fb_Product_Vacuum_Outlet_Isolation_Valve(Input1:= u01.product_vacuum_outlet_isolation_valve, Input2:= u.product_vacuum_outlet_isolation_valve, Output=> u01.XV_05);
u01.product_vacuum_outlet_isolation_valve_open_cmd_status				:= u01.XV_05;
u.product_vacuum_outlet_isolation_valve_clear							:= F_ValveClear(u.product_vacuum_outlet_isolation_valve, u01.product_vacuum_outlet_isolation_valve_open, u01.product_vacuum_outlet_isolation_valve_closed);

fb_Steam_Bypass_Valve(Input1:= u01.steam_bypass_valve, Input2:= u.steam_bypass_valve, Output=> u01.XV_08);
u01.steam_bypass_valve_open_cmd_status									:= u01.XV_08;
u.steam_bypass_valve_clear												:= F_ValveClear(u.steam_bypass_valve, u01.steam_bypass_valve_open, u01.steam_bypass_valve_closed);

fb_Condensate_Collection_Tank_Pump_Outlet_Valve(Input1:= u01.condensate_collection_tank_pump_outlet_valve, Input2:= u.condensate_collection_tank_pump_outlet_valve, Output=> );
u01.XV_09																:= u.condensate_collection_tank_pump_outlet_valve;
u01.condensate_collection_tank_pump_outlet_valve_open_cmd_status		:= u.condensate_collection_tank_pump_outlet_valve;
u.condensate_collection_tank_pump_outlet_valve_clear					:= F_ValveClear(u.condensate_collection_tank_pump_outlet_valve, u01.condensate_collection_tank_pump_outlet_valve_open, u01.condensate_collection_tank_pump_outlet_valve_closed);

fb_Product_Vacuum_Backfeed_Valve(Input1:= u01.product_vacuum_backfeed_valve, Input2:= u.product_vacuum_backfeed_valve);
fb_Product_Vacuum_Backfeed_Valve_Mode(Input1:= u01.product_vacuum_backfeed_valve_mode, Input2:= u.product_vacuum_backfeed_valve_mode);
fb_Product_Vacuum_Backfeed_Valve_PI(	Setpoint						:= u.product_vacuum_backfeed_valve_setpoint,
										Control							:= u01.product_vacuum_pres,
										Error							:= u01.product_vacuum_backfeed_valve_position_error,
										Reverse							:= FALSE,
										Kp								:= u01.product_vacuum_backfeed_valve_kp,           
										Ki								:= u01.product_vacuum_backfeed_valve_ki,           
										BaseAdjust						:= u01.product_vacuum_backfeed_valve_base_adjust,  
										LoopTime						:= u01.product_vacuum_backfeed_valve_loop_time,    
										IBand							:= u01.product_vacuum_backfeed_valve_iband,        
										Base							:= u01.product_vacuum_backfeed_valve_base,         
										Mode							:= u01.product_vacuum_backfeed_valve_mode,
										Input							:= u01.product_vacuum_backfeed_valve,
										Mode_Out						=> u01.product_vacuum_backfeed_valve_current_mode, 
										Output							=> u01.PCV_01);

u01.product_vacuum_backfeed_valve_position								:= INT_TO_REAL(u01.PCV_01_position) / _PERCENT_FACTOR; 
u.product_vacuum_backfeed_valve_open									:= u01.product_vacuum_backfeed_valve_position >= _VALVE_OPEN;
u01.product_vacuum_backfeed_valve_open									:= u.product_vacuum_backfeed_valve_open;
u.product_vacuum_backfeed_valve_closed									:= u01.product_vacuum_backfeed_valve_position < _VALVE_CLOSED;
u01.product_vacuum_backfeed_valve_closed								:= u.product_vacuum_backfeed_valve_closed;

fbSteamTotalizerEnable(Input1 := u01.steam_header_volume_total_enable, Input2 := u.steam_header_volume_total_enable );
//u01.steam_header_volume_total_enable 									:= u.steam_header_volume_total_enable;

fb_Product_Vacuum_Pump(					Enable							:= u01.product_vacuum_pump_vfd_enable,
										Pump_Reset						:= u01.product_vacuum_pump_reset,
										Purge_Time						:= u01.SP_product_vacuum_purge_time,
										Safety1							:= u01.P02_TSH_1,
										Safety2							:= u01.P02_TSH_2,
										Safety3							:= u01.P02_TSH_3,
										Error							=> u01.product_vacuum_pump_error,
										Purge_Solenoid_Valve			=> u01.P02_SVC_1,
										Seal_Purge_Valve				=> u01.P02_SVC_3);

sVacPumpError															:= CONCAT(gsProductVacuumPumpError, sVacuumPumpError[u01.product_vacuum_pump_error]);
bProductVacuumPumpError													:= P_Alarms.M_Check_Error(u01.product_vacuum_pump_error <> 0, bProductVacuumPumpError, _U01, sVacPumpError, gsProcessCannotRun);
						
fb_Product_Vacuum_Pump_Vfd_Input(Input1:= u01.product_vacuum_pump_vfd, Input2:= u.product_vacuum_pump_vfd);
rRpm																	:= u.product_vacuum_pump_vfd * _PUMP_RPM_FACTOR;
fb_Product_Vacuum_Pump_Vfd(				Enable_Vfd						:= fb_Product_Vacuum_Pump.Pump_On,
										Fault_Reset						:= u01.product_vacuum_pump_vfd_reset,
										Rpm								:= rRpm,
										Minimum_Speed					:= _PUMP_RPM_FACTOR * u01.SP_product_vacuum_idle_vfd_percent,
										Maximum_Speed					:= _PUMP_SPEED_MAX, 
										StatusWord						:= u01.product_vacuum_pump_vfd_status,
										ControlWord						=> u01.product_vacuum_pump_vfd_control, 
										TargetRpm						=> u01.product_vacuum_pump_vfd_target_vel, 
										Ready							=> u01.product_vacuum_pump_vfd_enabled,
										Error							=> u01.product_vacuum_pump_vfd_error);
u01.product_vacuum_pump_vfd_output  									:= WORD_TO_REAL(u01.product_vacuum_pump_vfd_velocity) / _PUMP_RPM_FACTOR ;                             
u.product_vacuum_pump_vfd_output										:= WORD_TO_REAL(u01.product_vacuum_pump_vfd_velocity);
IF u01.product_vacuum_pump_vfd_reset THEN
	u01.product_vacuum_pump_vfd_reset := FALSE;
END_IF

fb_Product_Vacuum_Pump_Radiator(Input1:= u01.radiator, Input2:= u.product_vacuum_pump_radiator);
u01.R_01																:= u.product_vacuum_pump_radiator;
u01.radiator_cmd_status													:= u.product_vacuum_pump_radiator;

// ignore if < 2 Amps
u01.l1_current_480														:= SEL(u01.IT_01 > _CURRENT_480_FACTOR * 2,0,F_IEConvert(u01.IT_01, _CURRENT_480_FACTOR));
u01.l2_current_480														:= SEL(u01.IT_02 > _CURRENT_480_FACTOR * 2,0,F_IEConvert(u01.IT_02, _CURRENT_480_FACTOR));
u01.l3_current_480														:= SEL(u01.IT_03 > _CURRENT_480_FACTOR * 2,0,F_IEConvert(u01.IT_03, _CURRENT_480_FACTOR));
u01.l1_voltage_480														:= F_IEConvert(u01.VT_01, _VOLTAGE_480_FACTOR);
u01.l2_voltage_480														:= F_IEConvert(u01.VT_02, _VOLTAGE_480_FACTOR);
u01.l3_voltage_480														:= F_IEConvert(u01.VT_03, _VOLTAGE_480_FACTOR);

// Ignore if < 1 Amp
u01.l1_current_208														:= SEL(u01.IT_04 > _CURRENT_208_FACTOR ,0,F_IEConvert(u01.IT_04, _CURRENT_208_FACTOR));
u01.l2_current_208														:= SEL(u01.IT_05 > _CURRENT_208_FACTOR ,0,F_IEConvert(u01.IT_05, _CURRENT_208_FACTOR));
u01.l3_current_208														:= SEL(u01.IT_06 > _CURRENT_208_FACTOR ,0,F_IEConvert(u01.IT_06, _CURRENT_208_FACTOR));
u01.l1_voltage_208														:= F_IEConvert(u01.VT_04, _VOLTAGE_208_FACTOR);
u01.l2_voltage_208														:= F_IEConvert(u01.VT_05, _VOLTAGE_208_FACTOR);
u01.l3_voltage_208														:= F_IEConvert(u01.VT_06, _VOLTAGE_208_FACTOR);

// Boiler - ignore noise if < 5A = 400 counts

u01.l1_current_boiler := SEL(u01.IT_boiler_01 > 400, 0, F_IEConvert(u01.IT_boiler_01, _CURRENT_BOILER_FACTOR));  // double coiled 
u01.l2_current_boiler := SEL(u01.IT_boiler_02 > 400, 0, F_IEConvert(u01.IT_boiler_02, _CURRENT_BOILER_FACTOR));  // double coiled 
u01.l3_current_boiler := SEL(u01.IT_boiler_03 > 400, 0, F_IEConvert(u01.IT_boiler_03, _CURRENT_BOILER_FACTOR));  // double coiled 

u01.boiler_ready														:= NOT u.boiler_outlet_pres_error AND u.boiler_outlet_pres > u01.SP_target_boiler_pressure AND u.boiler_package;
u.boiler_ready															:= u01.boiler_ready OR sita_bits[10].1;

tonBoilerCheck(IN:= u01.warmup_complete AND NOT u01.boiler_ready, PT:= _TIMEOUT_WARMUP_RESET);
IF tonBoilerCheck.Q THEN
	u01.warmup_complete													:= FALSE;
END_IF

// These Utility errors prevent any new automated cycles from running
u.utility_error															:= SEL(NOT u.boiler_ready, '', gsBoilerError);
u.utility_error															:= SEL(bDeadAirLinePresError, u.utility_error, gsDeadAirLinePresSensorError);		
u.utility_error															:= SEL(bPreCondenserLinePresError, u.utility_error, gsPreCondenserLinePresSensorError);
u.utility_error															:= SEL(bProductVacuumPresError, u.utility_error, gsProductVacuumPresSensorError);
u.utility_error															:= SEL(bProductVacuumPumpError, u.utility_error, gsProductVacuumPumpError);
u.utility_error															:= SEL(bProductOutletCo2Error, u.utility_error, gsProductOutletCo2SensorError);
u.utility_error															:= SEL(bProductOutletVolumetricFlowError, u.utility_error, gsProductOutletVolumetricFlowSensorError);
u.utility_error															:= SEL(bSteamHeaderFlowError, u.utility_error, gsSteamHeaderFlowSensorError);
u.utility_error															:= SEL(bBoilerOutletTempError, u.utility_error, gsBoilerOutletTempSensorError);
u.utility_error															:= SEL(bBoilerOutletPresError, u.utility_error, gsBoilerOutletPresSensorError);
u.utility_error															:= SEL(bProductCondensateDrumLevelError, u.utility_error, gsProductCondensateDrumLevelSensorError);
u.utility_error															:= SEL(bCondensateCollectionTankLevelError, u.utility_error, gsCondensateCollectionTankLevelSensorError);
u.utility_error															:= SEL(bWeatherTempUnsafe, u.utility_error, gsOutsideTempRangeError);
u.utility_error															:= SEL(bProductOutletPresError, u.utility_error, gsProductOutletPresSensorError);
u.utility_error															:= SEL(bProductOutletTempError, u.utility_error, gsProductOutletTempSensorError);
u.utility_error															:= SEL(bDeadAirLineCo2Error, u.utility_error, gsDeadAirLineCo2SensorError);
u.utility_error															:= SEL(bDeadAirFlowError, u.utility_error, gsDeadAirFlowSensorError);
u.utility_error															:= SEL(bProductOutletH2oError, u.utility_error, gsProductOutletH2oSensorError);
u.utility_error															:= SEL(bProductOutletO2Error, u.utility_error, gsProductOutletO2SensorError);
u.utility_error															:= SEL(bCondensateCollectionTankPhError, u.utility_error, gsCondensateCollectionTankPhSensorError);
u.utility_error															:= SEL(bCondensateCollectionTankO2Error, u.utility_error, gsCondensateCollectionTankO2SensorError);
u.utility_error															:= SEL(bCondensateCollectionTankTurbidityError, u.utility_error, gsCondensateCollectionTankTurbiditySensorError);
u.utility_error															:= SEL(bPurgeProductLinePresError, u.utility_error, gsPurgeProductLinePresSensorError);
u.utility_error															:= SEL(bPostCondenserLinePresError, u.utility_error, gsPostCondenserLinePresSensorError);
u.utility_error															:= SEL(bPurgeProductLineTempError, u.utility_error, gsPurgeProductLineTempSensorError);
u.utility_error															:= SEL(bPreCondenserLineTempError, u.utility_error, gsPreCondenserLineTempSensorError);
u.utility_error															:= SEL(bPostCondenserLineTempError, u.utility_error, gsPostCondenserLineTempSensorError);
u.utility_error															:= SEL(bProductCondenserPumpOutletTempError, u.utility_error, gsProductCondenserPumpOutletTempSensorError);
u.utility_error															:= SEL(bCondensateCollectionTankTempError, u.utility_error, gsCondensateCollectionTankTempSensorError);
u.utility_error															:= SEL(bCondensateCollectionTankOutletLineTempError, u.utility_error, gsCondensateCollectionTankOutletLineTempSensorError);
u.utility_error															:= SEL(bInstrumentAirCompPresError, u.utility_error, gsInstrumentAirCompPresSensorError);
u.utility_error															:= SEL(bInstrumentAirCompTempError, u.utility_error, gsInstrumentAirCompTempSensorError);
u.utility_error															:= SEL(bProductCondensateValveError, u.utility_error, gsProductCondensateDrainValveError);
sUtilityError															:= u.utility_error;

//P_Alarms.M_Add_Alarm('Utility', sUtilityError, 'Cycles_Stoppe');

// These errors initiate a Safe Shutdown if automated cycles are running 
IF m01.tb_Auto_Mode_On AND NOT bSafeShutdown THEN																			// Safe Shutdown 1
	u.safe_shutdown_error_1												:= SEL(bProductVacuumPumpError, '', gsProductVacuumPumpError);
	u.safe_shutdown_error_1												:= SEL(bPreCondenserLinePresError, u.safe_shutdown_error_1, gsPreCondenserLinePresSensorError);
	u.safe_shutdown_error_1												:= SEL(bProductVacuumPresError, u.safe_shutdown_error_1, gsProductVacuumPresSensorError);
	u.safe_shutdown_error_1												:= SEL(bProductOutletCo2Error, u.safe_shutdown_error_1, gsProductOutletCo2SensorError);
	u.safe_shutdown_error_1												:= SEL(bProductOutletVolumetricFlowError, u.safe_shutdown_error_1, gsProductOutletCo2SensorError);
	IF u.safe_shutdown_error_1 <> '' THEN
		bSafeShutdown													:= TRUE;
	ELSE																													// Safe Shutdown 2
		u.safe_shutdown_error_2											:= SEL(bSteamHeaderFlowError, '', gsSteamHeaderFlowSensorError);
		u.safe_shutdown_error_2											:= SEL(bBoilerOutletPresError, u.safe_shutdown_error_2, gsBoilerOutletPresSensorError);
		u.safe_shutdown_error_2											:= SEL(bBoilerOutletTempError, u.safe_shutdown_error_2, gsBoilerOutletTempSensorError);
		u.safe_shutdown_error_2											:= SEL(NOT u.boiler_ready, u.safe_shutdown_error_2, gsBoilerError);
		u.safe_shutdown_error_2											:= SEL(P_M01.bSteamManifoldLinePresError, u.safe_shutdown_error_2, gsSteamManifoldLinePresSensorError);
		u.safe_shutdown_error_2											:= SEL(P_M01.bSteamTempNearRS01Error, u.safe_shutdown_error_2, gsSteamTempNearRS01SensorError);
		u.safe_shutdown_error_2											:= SEL(P_M01.bSteamTempNearRS03Error, u.safe_shutdown_error_2, gsSteamTempNearRS03SensorError);
		u.safe_shutdown_error_2											:= SEL(bProductCondensateDrumLevelError, u.safe_shutdown_error_2, gsProductCondensateDrumLevelSensorError);
		u.safe_shutdown_error_2											:= SEL(bCondensateCollectionTankLevelError, u.safe_shutdown_error_2, gsCondensateCollectionTankLevelSensorError);
		IF u.safe_shutdown_error_2 <> '' THEN
			bSafeShutdown												:= TRUE;
		END_IF
	END_IF
ELSIF NOT m01.tb_Auto_Mode_On THEN
	bSafeShutdown														:= FALSE;
	u.safe_shutdown_error_1												:= '';
	u.safe_shutdown_error_2												:= '';
END_IF
END_ACTION

ACTION A_Totalizers:
tmrTotalizers(IN := NOT tmrTotalizers.Q,PT := T#1S);
// get steam density every 1 sec  
IF tmrTotalizers.Q THEN
	
 // Steam volume
	FOR idxSteamTable := 1 TO 30 DO 
		IF u01.boiler_outlet_pres >= STEAM_TABLE[idxSteamTable][0] THEN
			rSteamDensity := STEAM_TABLE[idxSteamTable][1];
		END_IF
	END_FOR
	
    u01.steam_header_volume := rSteamDensity * (u01.steam_header_flow*1000)/60 * 1.0;  // density kg/l  * flow m3/min ( m3 = 1000l)  * 1 sec 
	IF u01.steam_header_volume_total_enable THEN
		u01.steam_header_volume_total := u01.steam_header_volume_total + u01.steam_header_volume;
	ELSE
		u01.steam_header_volume_total := 0;
	END_IF
	
	// Product flows 
	IF u01.product_outlet_mass_flow_total_enable OR u01.product_outlet_volumetric_flow_total_enable THEN 
		u01.product_outlet_mass_flow_total := u01.product_outlet_mass_flow_total + u01.product_outlet_mass_flow/60 * 1.0;  //  kg/min to kg/sec * 1 sec
		u01.product_outlet_volumetric_flow_total := u01.product_outlet_volumetric_flow_total + u01.product_outlet_volumetric_flow/60 * 1.0 ;  // l/min to t/sec  * 1 sec
	ELSE
		u01.product_outlet_mass_flow_total := 0;
		u01.product_outlet_volumetric_flow_total := 0;
	END_IF
	
	// Bolier Water flow 
	
	IF u01.tap_water_to_boiler_flow_total_enable THEN 
		u01.tap_water_to_boiler_flow_total := u01.tap_water_to_boiler_flow_total +  u01.tap_water_to_boiler_flow/60 * 1.0; // //  kg/min to kg/sec * 1 sec
	ELSE
		u01.tap_water_to_boiler_flow_total := 0;
	END_IF
 
END_IF
END_ACTION

ACTION A_Weather_Station:
// Phase 0 - A_Weather_Station
// Rev 1.00 - February 5, 2024

IF iWSFunction = 0 THEN																		// Modbus is not busy
	WS_Master.UnitID 													:= 1;				// Weather Station Modbus address
	wWSAddress															:= 8193;
	wWSQuantity															:= 1;
	iWSFunction															:= eWSReadRegs;
	// Get weather values here
	//	ZXI_2002														:= wMBPReadData[0];
	//	ZYI_2002														:= wMBPReadData[1];
ELSIF tonWSReset.Q THEN
	iWSFunction															:= eWSIdle;
END_IF
tonWSReset(IN:= iWSFunction > 0, PT:= _TIMEOUT_MODBUS);

CASE iWSFunction OF
	
	eWSIdle:
		WS_Master.Execute 												:= FALSE;
		
	eWSReadRegs:
		WS_Master.ReadRegs(		Quantity								:= wWSQuantity, 
								MBAddr									:= wWSAddress, 
								cbLength								:= SIZEOF(wWSReadData), 
								pMemoryAddr								:= ADR(wWSReadData), 
								Execute									:= TRUE, 
								Timeout									:= _TIMEOUT_MODBUS, 
								BUSY									=> bWSBusy, 
								Error									=> bWSError, 
								ErrorId									=> WS_Errors, 
								cbRead									=> uiWSRead);
			
		WS_Master.ReadRegs(BUSY=> bWSBusy);
		IF NOT WS_Master.BUSY THEN
			WS_Master.Execute 											:= FALSE;
			WS_Master.ReadRegs(BUSY=> bWSBusy);
			IF WS_Master.Error THEN
				WS_Master.ReadRegs();
			ELSE
				iWSFunction 											:= 0;			
			END_IF
		END_IF
	
	ELSE
		iWSFunction 													:= 0;
	
END_CASE
END_ACTION

ACTION A2_WarmUp:
// Phase 0 - P_U01.A2_WarmUp
// Rev 1.0 - April 4, 2024

CASE i2Step OF

	0:	;
		
	1:	
		sError															:= '';
		bComplete														:= FALSE;
		bRunSteamBypass													:= FALSE;
		u01.steam_bypass_complete										:= FALSE;
		IF NOT u01.warmup_complete THEN
			gsCycleStage												:= 'warm_up.initialize';							// 3
			IF u01.boiler_outlet_pres_error THEN
				sError													:= F_Concat3(_U01, gsCycleStage, gsBoilerError);
				i2Step													:= 80;
			ELSE
				i2Step													:= i2Step + 1;
			END_IF
		ELSE
			bComplete													:= TRUE;
			i2Step														:= 90;
		END_IF
		
	2:	
		u01.boiler_package												:= TRUE;											// 4
		gsCycleStage													:= 'warm_up.boiler_heating';						// 5
		u01.drainage_on													:= TRUE;											// 6
		bAdsorptionActive												:= FALSE;											// 7
		bAdsorptionTimer												:= FALSE;
		i2Step															:= SEL(u01.SP_adsorb_during_warmup, 20, i2Step + 1);	// 8

	3:
		iAxStep															:= 1;												// 8.a
		i2Step															:= i2Step + 1;

	4:	
		Ax_Process_Pre_Check();																								// 8.a																			
		IF bPreCheckDone THEN
			IF sError = '' THEN																								// 8.a.i
				P_M01_RS01.open_repres_valves							:= P_M01.bRS01;										// 8.b
				P_M01_RS02.open_repres_valves							:= P_M01.bRS02;
				P_M01_RS03.open_repres_valves							:= P_M01.bRS03;
				rTime													:= _VALVE_TIME;
				i2Step													:= i2Step + 1;
			ELSE
				P_Alarms.M_Add_Alarm(CONCAT(_U01, gsCycleStage), sError, gsWarmupWillContinueWOAdsorption);					// 8.a.ii
				i2Step													:= 20;
			END_IF
		END_IF
		
	5:
		bTimer															:= TRUE;
		bPass1															:= (P_M01.bRS01 AND P_M01_RS01.repres_valves_clear) OR NOT P_M01.bRS01;
		bPass2															:= (P_M01.bRS02 AND P_M01_RS02.repres_valves_clear) OR NOT P_M01.bRS02;
		bPass3															:= (P_M01.bRS03 AND P_M01_RS03.repres_valves_clear) OR NOT P_M01.bRS03;
		IF bPass1 AND bPass2 AND bPass3 THEN
			bTimer														:= FALSE;
			i2Step														:= i2Step + 1;
		ELSIF tonTimer.Q THEN
			bTimer														:= FALSE;
			//P_M01_RS01.close_repres_valves								:= TRUE;
			//P_M01_RS02.close_repres_valves								:= TRUE;
			//P_M01_RS03.close_repres_valves								:= TRUE;
			//P_Alarms.M_Add_Alarm(CONCAT(_U01, gsCycleStage), M_Repres_Valve_Error(), gsWarmupWillContinueWOAdsorption);	// Per Alex W.
			//i2Step														:= 20;
			i2Step														:= i2Step + 1; 
		END_IF
		
	6:
		P_M01_RS01.open_all_doors										:= P_M01.bRS01;										// 8.c
		P_M01_RS02.open_all_doors										:= P_M01.bRS02;
		P_M01_RS03.open_all_doors										:= P_M01.bRS03;
		rTime															:= m01.SP_doorsopenclose_timedelay * _MINUTES;										// 8.c.i
		gsCycleStage													:= 'warm_up.boiler_heating_open_doors';				// 8.c.ii
		i2Step															:= i2Step + 1;

	7:
		bTimer															:= TRUE; 
		bPass1															:= (P_M01.bRS01 AND P_M01_RS01.R_S.all_doors_open) OR NOT P_M01.bRS01;
		bPass2															:= (P_M01.bRS02 AND P_M01_RS02.R_S.all_doors_open) OR NOT P_M01.bRS02;
		bPass3															:= (P_M01.bRS03 AND P_M01_RS03.R_S.all_doors_open) OR NOT P_M01.bRS03;
		IF bPass1 AND bPass2 AND bPass3 THEN
			bTimer														:= FALSE;
			i2Step														:= i2Step + 1;
		ELSIF tonTimer.Q THEN
			bTimer														:= FALSE;
			sRS															:= SEL(NOT bPass1, SEL(NOT bPass2, _RS03, _RS02), _RS01);
			P_Alarms.M_Add_Alarm(F_Concat3(_U01, sRS, gsCycleStage), gsReactorDoorOpeningError, gsWarmupWillContinueWOAdsorption);
			i2Step														:= 20;
		END_IF

	8:
		P_M01_RS01.fan_vfd_percent										:= SEL(P_M01.bRS01, 0, m01.SP_reactor_set_1_vfd_percent);	// 8.d
		P_M01_RS02.fan_vfd_percent										:= SEL(P_M01.bRS02, 0, m01.SP_reactor_set_2_vfd_percent);
		P_M01_RS03.fan_vfd_percent										:= SEL(P_M01.bRS03, 0, m01.SP_reactor_set_3_vfd_percent);
		gsCycleStage													:= 'warm_up.boiler_heating_turn_on_fans';			// 8.d.i
		rTime															:= _FAN_RS_DELAY_TIME;
		i2Step															:= i2Step + 1;

	9:
		bTimer															:= TRUE;
		IF tonTimer.Q THEN
			bTimer														:= FALSE;
			i2Step														:= i2Step + 1;
		END_IF

	10:
		P_M01_RS01.co2_inside_sensors_on								:= P_M01.bRS01;										// 8.e
		P_M01_RS02.co2_inside_sensors_on								:= P_M01.bRS02;
		P_M01_RS03.co2_inside_sensors_on								:= P_M01.bRS03;
		gsCycleStage													:= 'warm_up.boiler_heating_adsorption';				// 8.e.i
		bAdsorptionTimer												:= TRUE;											// 8.f
		bAdsorptionActive												:= TRUE;											// 8.g
		i2Step															:= 20;


//**** Complete Warmup		
	20:
		u01.product_vacuum_backfeed_valve								:= _OPEN;											// 9
		rTime															:= _VALVE_TIME;
		i2Step															:= i2Step + 1;
		
	21:	
		bTimer															:= TRUE;
		IF u01.product_vacuum_backfeed_valve_open THEN																		// 9
			bTimer														:= FALSE;
			u01.product_vacuum_pump_vfd									:= u01.SP_product_vacuum_idle_vfd_percent;			// 10
			rTime														:= u01.SP_boiler_warmup_duration * _MINUTES;		// 11
			i2Step														:= i2Step + 1;
		ELSIF tonTimer.Q THEN
			bTimer														:= FALSE;
			sError														:= gsProductVacuumBackfeedValveError;				// 9
			IF bAdsorptionActive THEN
				P_Alarms.M_Add_Alarm(CONCAT(_U01, gsCycleStage), sError, gsProcessCannotRunAdsorptionWillContinue);
				u01.boiler_package										:= FALSE;
				i2Step													:= 30;
			ELSE
				i2Step													:= 80;
			END_IF
		END_IF
		
	22:
		bTimer															:= TRUE;
		IF u01.boiler_ready THEN																							// 12 (Handled in P_U01.A_Points)
			bTimer														:= FALSE;
			bComplete													:= TRUE;
			u01.warmup_complete											:= TRUE;
			i2Step														:= i2Step + 1;
		ELSIF tonTimer.Q THEN																								// 12.a
			bTimer														:= FALSE;
			sError														:= gsBoilerError;
			i2Step														:= 80;
		END_IF

	23:
		bRunSteamBypass													:= u01.SP_steam_bypass_immediately_after_warm_up;
		IF bAdsorptionActive AND NOT bRunSteamBypass THEN 																	// 14
			i2Step														:= 30;
		ELSIF bAdsorptionActive AND bRunSteamBypass AND NOT u01.SP_adsorb_during_steam_bypass THEN
			i2Step														:= 40;												// 15
		ELSE
			i2Step														:= 90;												// 13 & 16
		END_IF
	
		
//**** Adsorption 1		
	30:
		IF tonAdsorptionTimer.Q THEN																						// 14.a
			bAdsorptionTimer											:= FALSE;
			gsCycleStage												:= 'warm_up.boiler_heating.turn_off_fans';			// 14.b
			P_M01_RS01.fan_vfd_percent									:= 0;												// 14.c
			P_M01_RS02.fan_vfd_percent									:= 0;
			P_M01_RS03.fan_vfd_percent									:= 0;
			rTime														:= _FAN_RS_DELAY_TIME;
			i2Step														:= i2Step + 1;
		END_IF

	31:
		bTimer															:= TRUE;
		IF tonTimer.Q THEN
			bTimer														:= FALSE;
			gsCycleStage												:= 'warm_up.boiler_heating.closing_doors';			// 14.d
			P_M01_RS01.close_all_doors									:= TRUE;											// 14.e
			P_M01_RS02.close_all_doors									:= TRUE;
			P_M01_RS03.close_all_doors									:= TRUE;
			rTime														:= m01.SP_doorsopenclose_timedelay * _MINUTES;										// 14.e.i
			i2Step														:= i2Step + 1;
		END_IF		

	32:
		bTimer															:= TRUE;
		bPass1															:= (P_M01.bRS01 AND P_M01_RS01.R_S.all_doors_closed) OR NOT P_M01.bRS01;	// 14.e.ii
		bPass2															:= (P_M01.bRS02 AND P_M01_RS02.R_S.all_doors_closed) OR NOT P_M01.bRS02;
		bPass3															:= (P_M01.bRS03 AND P_M01_RS03.R_S.all_doors_closed) OR NOT P_M01.bRS03;
		IF bPass1 AND bPass2 AND bPass3 THEN
			bTimer														:= FALSE;
			i2Step														:= i2Step + 1;
		ELSIF tonTimer.Q THEN																								// 14.e.i
			bTimer														:= FALSE;
			bRunSteamBypass												:= FALSE;
			sRS															:= SEL(NOT bPass1, SEL(NOT bPass2, _RS03, _RS02), _RS01);
			P_Alarms.M_Add_Alarm(F_Concat3(_U01, sRS, gsCycleStage), gsReactorDoorClosingError, gsSystemCannotRun);
			i2Step														:= i2Step + 1;
		END_IF
		
	33:
		P_M01_RS01.co2_sensors_off										:= TRUE;											// 14.f
		P_M01_RS02.co2_sensors_off										:= TRUE;
		P_M01_RS03.co2_sensors_off										:= TRUE;
		bAdsorptionActive												:= FALSE;											// 14.g
		i2Step															:= 90;

	
//**** Adsorption 2	
	40:
		IF tonAdsorptionTimer.Q THEN																						// 15.a
			bAdsorptionTimer											:= FALSE;
			P_M01_RS01.fan_vfd_percent									:= 0;												// 15.b
			P_M01_RS02.fan_vfd_percent									:= 0;
			P_M01_RS03.fan_vfd_percent									:= 0;
			rTime														:= _FAN_RS_DELAY_TIME;
			i2Step														:= i2Step + 1;
		END_IF

	41:
		bTimer															:= TRUE;
		IF tonTimer.Q THEN
			bTimer														:= FALSE;											// 15.c
			P_M01_RS01.co2_sensors_off									:= TRUE;
			P_M01_RS02.co2_sensors_off									:= TRUE;
			P_M01_RS03.co2_sensors_off									:= TRUE;
			bAdsorptionActive											:= FALSE;											// 15.d
			i2Step														:= i2Step + 1;
		END_IF
		
	42:
		P_M01_RS01.close_all_doors										:= TRUE;											// 15.g
		P_M01_RS02.close_all_doors										:= TRUE;
		P_M01_RS03.close_all_doors										:= TRUE;
		rTime															:= m01.SP_doorsopenclose_timedelay * _MINUTES;										// 15.g.i
		i2Step															:= i2Step + 1;

	43:
		bTimer															:= TRUE;
		bPass1															:= (P_M01.bRS01 AND P_M01_RS01.R_S.all_doors_closed) OR NOT P_M01.bRS01;		// 15.g.ii
		bPass2															:= (P_M01.bRS02 AND P_M01_RS02.R_S.all_doors_closed) OR NOT P_M01.bRS02;
		bPass3															:= (P_M01.bRS03 AND P_M01_RS03.R_S.all_doors_closed) OR NOT P_M01.bRS03;
		IF bPass1 AND bPass2 AND bPass3 THEN
			bTimer														:= FALSE;
			i2Step														:= 90;
		ELSIF tonTimer.Q THEN
			bTimer														:= FALSE;
			bRunSteamBypass												:= FALSE;
			sRS															:= SEL(NOT bPass1, SEL(NOT bPass2, _RS03, _RS02), _RS01);
			P_Alarms.M_Add_Alarm(F_Concat3(_U01, sRS, gsCycleStage), gsReactorDoorOpeningError, gsSystemCannotRun);
			i2Step														:= 90;
		END_IF


//**** Process error		
	80:
		P_Alarms.M_Add_Alarm(CONCAT(_U01, gsCycleStage), sError, gsProcessCannotRun);
		gsCycleStage													:= 'warm_up.error';
		i2Step															:= i2Step + 1;

//**** Stop process		
	81:
		u01.product_vacuum_pump_vfd										:= 0;
		u01.product_vacuum_backfeed_valve								:= _CLOSED;
		P_M01_RS01.co2_sensors_off										:= TRUE;
		P_M01_RS02.co2_sensors_off										:= TRUE;
		P_M01_RS03.co2_sensors_off										:= TRUE;
		P_M01_RS01.fan_vfd_percent										:= 0;
		P_M01_RS02.fan_vfd_percent										:= 0;
		P_M01_RS03.fan_vfd_percent										:= 0;
		rTime															:= _FAN_RS_DELAY_TIME;
		i2Step															:= i2Step + 1;

	82:
		bTimer															:= TRUE;
		IF tonTimer.Q THEN
			bTimer														:= FALSE;
			u01.boiler_package											:= FALSE;
			P_M01_RS01.close_all_doors									:= P_M01.bRS01;
			P_M01_RS02.close_all_doors									:= P_M01.bRS02;
			P_M01_RS03.close_all_doors									:= P_M01.bRS03;
			rTime														:= m01.SP_doorsopenclose_timedelay * _MINUTES;
			i2Step														:= 90;
		END_IF
		
//**** Close process
	90:
		gsCycleStage													:= SEL(bComplete, 'warm_up.failed', 'warm_up.complete');
		bAdsorptionTimer												:= FALSE;
		u01.drainage_on													:= FALSE;
		rTime															:= _PROCESS_COMPLETE_TIME;
		i2Step															:= i2Step + 1;
		
	91:
		bTimer															:= TRUE;
		IF tonTimer.Q THEN
			bTimer														:= FALSE;
			gsCycleStage												:= '';
			i2Step														:= 0;
		END_IF
				

END_CASE

IF i2Step > 0 AND i2Step < 80 AND u01.shutdown_process THEN
	gsCycleStage														:= 'warm_up.stopping';
	i2Step																:= 81;
END_IF
END_ACTION

ACTION A3_Steam_Bypass:
// Phase 0 - P_U01.A3_Steam_Bypass
// Rev 1.0 - April 4, 2024

CASE i3Step OF

	0:	;

	1:	
		bComplete														:= FALSE;
		IF u01.warmup_complete THEN
			IF NOT u01.steam_bypass_complete THEN
				gsCycleStage											:= 'steam_bypass.initialize';						// 4
				sError													:= '';
				IF u01.post_condenser_line_pres_error THEN
					sError												:= gsPostCondenserLinePresSensorError;
				ELSIF u01.pre_condenser_line_pres_error THEN
					sError												:= gsPreCondenserLinePresSensorError;
				ELSIF u01.purge_product_line_pres_error THEN
					sError												:= gsPurgeProductLinePresSensorError;
				ELSIF u01.product_vacuum_pres_error THEN
					sError												:= gsProductVacuumPresSensorError;
				ELSIF u01.steam_header_flow_error THEN
					sError												:= gsSteamHeaderFlowSensorError;
				ELSIF u01.purge_product_line_temp_error THEN
					sError												:= gsPurgeProductLineTempSensorError;
				END_IF
				i3Step													:= SEL(sError = '', 80, i3Step + 1);
			ELSE
				bComplete												:= TRUE;
				i3Step													:= 90;
			END_IF
		ELSE
			u01.boiler_package											:= FALSE;
			P_Alarms.M_Add_Alarm(CONCAT(_U01, gsCycleStage), gsWarmupNotRunError, gsProcessCannotRun);
			i3Step														:= 90;
		END_IF
		
	2:	
		IF u01.boiler_ready THEN																							// 5.a (Handled in P_U01.A_Points)
			P_U01.bCloseXVValves										:= TRUE;											// 5.b
			rTime														:= _VALVE_TIME;
			i3Step														:= i3Step + 1;
		ELSE
			sError														:= gsBoilerError;
			sMessage													:= gsRunWarmup;
			i3Step														:= 80;
		END_IF

	3:	bTimer															:= TRUE;
		bPass1															:= u01.product_vacuum_pump_isolation_valve_closed;
		bPass2															:= u01.product_vacuum_outlet_isolation_valve_closed;
		IF bPass1 AND bPass2 THEN
			bTimer														:= FALSE;
			u01.product_vacuum_backfeed_valve							:= _OPEN;											// 5.b.iii
			rTime														:= _VALVE_TIME;
			i3Step														:= i3Step + 1;
		ELSIF tonTimer.Q THEN
			bTimer														:= FALSE;
			sError														:= SEL(bPass1, '', gsProductVacuumPumpIsoValveError);
			sError														:= SEL(bPass2, sError, gsProductVacuumOutletIsoValveError);
			i3Step														:= 80;
		END_IF
		
	4:
		bTimer															:= TRUE;
		IF u01.product_vacuum_backfeed_valve > _VALVE_OPEN THEN
			bTimer														:= FALSE;
			u01.drainage_on												:= TRUE;											// 5.c
			u01.product_vacuum_pump_vfd									:= u01.SP_product_vacuum_idle_vfd_percent;			// 5.d.ii
			IF bAdsorptionActive AND u01.SP_adsorb_during_steam_bypass THEN													// 5.b.iv
				P_M01_RS01.open_all_doors								:= P_M01.bRS01;
				P_M01_RS02.open_all_doors								:= P_M01.bRS02;
				P_M01_RS03.open_all_doors								:= P_M01.bRS03;
				rTime													:= m01.SP_doorsopenclose_timedelay * _MINUTES;
				i3Step													:= i3Step + 1;
			ELSE
				i3Step													:= i3Step + 2;
			END_IF
		ELSIF tonTimer.Q THEN
			bTimer														:= FALSE;
			sError														:= gsProductVacuumBackfeedValveError;
			i3Step														:= 80;
		END_IF

	5:
		bTimer															:= TRUE;
		bPass1															:= (P_M01.bRS01 AND P_M01_RS01.R_S.all_doors_open) OR NOT P_M01.bRS01;	// 5.b.iv
		bPass2															:= (P_M01.bRS02 AND P_M01_RS02.R_S.all_doors_open) OR NOT P_M01.bRS02;
		bPass3															:= (P_M01.bRS03 AND P_M01_RS03.R_S.all_doors_open) OR NOT P_M01.bRS03;
		IF bPass1 AND bPass2 AND bPass3 THEN
			bTimer														:= FALSE;
			IF NOT bAdsorptionActive AND u01.SP_adsorb_during_steam_bypass THEN												// 6
				iAxStep													:= 1;												// 6.b
				i3Step													:= i3Step + 1;
			ELSE
				i3Step													:= 20;
			END_IF
		ELSIF tonTimer.Q THEN
			bTimer														:= FALSE;
			bAdsorptionActive											:= FALSE;
			sRS															:= SEL(NOT bPass1, SEL(NOT bPass2, _RS03, _RS02), _RS01);
			P_Alarms.M_Add_Alarm(F_Concat3(_U01, sRS, gsCycleStage), gsReactorDoorOpeningError, gsSteamBypassWillContinueWOAdsorption);
			i3Step														:= 20;
		END_IF

	6:
		Ax_Process_Pre_Check();																								// 6.b																			
		IF bPreCheckDone THEN
			IF sError = '' THEN																								// 6.b.i
				P_M01_RS01.open_repres_valves							:= P_M01.bRS01;										// 6.c
				P_M01_RS02.open_repres_valves							:= P_M01.bRS02;
				P_M01_RS03.open_repres_valves							:= P_M01.bRS03;
				rTime													:= _VALVE_TIME;
				i3Step													:= i3Step + 1;
			ELSE
				P_Alarms.M_Add_Alarm(CONCAT(_U01, gsCycleStage), sError, gsSteamBypassWillContinueWOAdsorption);			// 6.b.ii
				bAdsorptionActive										:= FALSE;
				i3Step													:= 20;
			END_IF
		END_IF

	7:
		bTimer															:= TRUE;
		bPass1															:= (P_M01.bRS01 AND P_M01_RS01.repres_valves_clear) OR NOT P_M01.bRS01;
		bPass2															:= (P_M01.bRS02 AND P_M01_RS02.repres_valves_clear) OR NOT P_M01.bRS02;
		bPass3															:= (P_M01.bRS03 AND P_M01_RS03.repres_valves_clear) OR NOT P_M01.bRS03;
		IF bPass1 AND bPass2 AND bPass3 THEN
			bTimer														:= FALSE;
			i3Step														:= i3Step + 1;
		ELSIF tonTimer.Q THEN
			bTimer														:= FALSE;
			i3Step														:= i3Step + 1;
			//P_Alarms.M_Add_Alarm(CONCAT(_U01, gsCycleStage), M_Repres_Valve_Error(), gsSteamBypassWillContinueWOAdsorption);
			//bAdsorptionActive											:= FALSE;
			//P_M01_RS01.close_repres_valves								:= P_M01.bRS01;
			//P_M01_RS02.close_repres_valves								:= P_M01.bRS02;
			//P_M01_RS03.close_repres_valves								:= P_M01.bRS03;
			//i3Step													:= 20; 
		END_IF
		
	8:
		P_M01_RS01.open_all_doors										:= P_M01.bRS01;
		P_M01_RS02.open_all_doors										:= P_M01.bRS02;
		P_M01_RS03.open_all_doors										:= P_M01.bRS03;
		gsCycleStage													:= 'steam_bypass.initialize.open_doors';			// 6.d.ii
		rTime															:= m01.SP_doorsopenclose_timedelay * _MINUTES;										// 6.d.i
		i3Step															:= i3Step + 1;

	9:
		bTimer															:= TRUE; 
		bPass1															:= (P_M01.bRS01 AND P_M01_RS01.R_S.all_doors_open) OR NOT P_M01.bRS01;	// 6.d.ii
		bPass2															:= (P_M01.bRS02 AND P_M01_RS02.R_S.all_doors_open) OR NOT P_M01.bRS02;
		bPass3															:= (P_M01.bRS03 AND P_M01_RS03.R_S.all_doors_open) OR NOT P_M01.bRS03;
		IF bPass1 AND bPass2 AND bPass3 THEN
			bTimer														:= FALSE;
			i3Step														:= i3Step + 1;
		ELSIF tonTimer.Q THEN
			bTimer														:= FALSE;
			sRS															:= SEL(NOT bPass1, SEL(NOT bPass2, _RS03, _RS02), _RS01);
			P_Alarms.M_Add_Alarm(F_Concat3(_U01, sRS, gsCycleStage), gsReactorDoorOpeningError, gsSteamBypassWillContinueWOAdsorption);
			bAdsorptionActive											:= FALSE;
			i3Step														:= 20;
		END_IF

	10:
		P_M01_RS01.fan_vfd_percent										:= SEL(P_M01.bRS01, 0, m01.SP_reactor_set_1_vfd_percent);	// 6.e
		P_M01_RS02.fan_vfd_percent										:= SEL(P_M01.bRS02, 0, m01.SP_reactor_set_2_vfd_percent);
		P_M01_RS03.fan_vfd_percent										:= SEL(P_M01.bRS03, 0, m01.SP_reactor_set_3_vfd_percent);
		gsCycleStage													:= 'steam_bypass.initialize.turn_on_fans';			// 6.e.i
		rTime															:= _FAN_RS_DELAY_TIME;
		i3Step															:= i3Step + 1;

	11:
		bTimer															:= TRUE;
		IF tonTimer.Q THEN
			bTimer														:= FALSE;
			i3Step														:= i3Step + 1;
		END_IF

	12:
		P_M01_RS01.co2_inside_sensors_on								:= P_M01.bRS01;										// 6.f
		P_M01_RS02.co2_inside_sensors_on								:= P_M01.bRS02;
		P_M01_RS03.co2_inside_sensors_on								:= P_M01.bRS03;
		gsCycleStage													:= 'steam_bypass.initialize.adsorption';			// 6.f.i
		bAdsorptionTimer												:= TRUE;											// 6.a
		bAdsorptionActive												:= TRUE;											// 6.g
		i3Step															:= 20;


//**** Complete Steam Bypass		
	20:
		u01.product_condenser											:= TRUE;											// 7
		rSP																:= u01.SP_steam_bypass_vacuum_pressure;				// 8
		bPass1															:= u01.product_vacuum_pres < rSP;
		bPass2															:= u01.post_condenser_line_pres < rSP;
		bPass3															:= u01.pre_condenser_line_pres < rSP;
		bPass4															:= u01.purge_product_line_pres < rSP;
		i3Step															:= SEL(bPass1 AND bPass2 AND bPass3 AND bPass4, i3Step + 1, 30);
	
	21:
		u01.product_vacuum_pump_isolation_valve							:= TRUE;											// 9.a
		u01.product_vacuum_outlet_isolation_valve						:= TRUE;
		rTime															:= _VALVE_TIME;
		i3Step															:= i3Step + 1;
		
	22:
		bTimer															:= TRUE;
		bPass1															:= u01.product_vacuum_pump_isolation_valve_open;
		bPass2															:= u01.product_vacuum_outlet_isolation_valve_open;
		IF bPass1 AND bPass2 THEN
			bTimer														:= FALSE;
			//u01.product_blower											:= TRUE;											// 9.a
			u.product_blower_vfd										:= 0;  //
			u01.product_vacuum_backfeed_valve							:= _CLOSED;
			i3Step														:= i3Step + 1;
		ELSIF tonTimer.Q THEN
			bTimer														:= FALSE;
			sError														:= SEL(bPass1, '', gsProductVacuumPumpIsoValveError);
			sError														:= SEL(bPass2, sError, gsProductVacuumOutletIsoValveError);
			i3Step														:= 80;
		END_IF
		
	23:	
		u01.product_vacuum_pump_vfd										:= u01.SP_product_vacuum_running_vfd_percent;			// 9.b
		gsCycleStage													:= SEL(bAdsorptionActive, 'steam_bypass.evacuate_lines', 'steam_bypass.evacuate_lines.adsorption');		// 9.b.i
		u01.purge_product_pre_condenser_valve							:= TRUE;											// 9.c
		u01.cooling_line_pre_condenser_valve							:= TRUE;
		rTime															:= m01.SP_evacuation_duration * _MINUTES;
		i3Step															:= i3Step + 1;
		
	24:
		bTimer															:= TRUE;											// 9.d
		rSP																:= u01.SP_steam_bypass_vacuum_pressure;
		bPass1															:= u01.product_vacuum_pres < rSP;
		bPass2															:= u01.post_condenser_line_pres < rSP;
		bPass3															:= u01.pre_condenser_line_pres < rSP;
		bPass4															:= u01.purge_product_line_pres < rSP;
		IF bPass1 AND bPass2 AND bPass3 AND bPass4 THEN
			bTimer														:= FALSE;
			i3Step														:= i3Step + 1;
		ELSIF tonTimer.Q THEN
			bTimer														:= FALSE;
			sError														:= gsUnableToEvacuateLinesError;
			i3Step														:= 80;
		END_IF
	
	25:	
		u01.product_vacuum_pump_isolation_valve							:= FALSE;											// 9.e
		u01.product_vacuum_outlet_isolation_valve						:= FALSE;
		u01.product_vacuum_backfeed_valve								:= _OPEN;
		//u01.product_blower											:= FALSE;
		u.product_blower_vfd											:= 0;
		u01.cooling_line_pre_condenser_valve							:= FALSE;
		u01.purge_product_pre_condenser_valve							:= FALSE;
		u01.product_vacuum_pump_vfd										:= u01.SP_product_vacuum_idle_vfd_percent;			// 9.f
		i3Step															:= 30;

		
//**** Steam Bypass		
	30:
		u01.steam_bypass_valve											:= TRUE;											// 10
		gsCycleStage													:= SEL(bAdsorptionActive, 'steam_bypass.steam_bypass.adsorption', 'steam_bypass.steam_bypass');		// 10.a
		rSP																:= u01.SP_steam_bypass_duration * _MINUTES;				
		rTime															:= rSP;
		i3Step															:= i3Step + 1;				

	31:
		bTimer															:= TRUE;											// 10.b
		IF u01.purge_product_line_pres > m01.SP_steam_purge_pressure THEN													// 11
			i3Step														:= i3Step + 1;
		ELSIF tonTimer.Q THEN
			bTimer														:= FALSE;
			sError														:= gsPurgeProductLinePresLowError;
			i3Step														:= 80;
		END_IF
		
	32:
		u01.product_vacuum_bypass_valve									:= TRUE;											// 12
		u01.purge_product_pre_condenser_valve							:= TRUE;
		//u01.product_blower												:= TRUE;
		u.product_blower_vfd											:= _BLOWER_RPM_FACTOR * 100; // % TBD 
		i3Step															:= i3Step + 1;
		
	33:
		IF TIME_TO_REAL(tonTimer.ET) >= (rSP * 0.3) THEN																	// 13
			i3Step														:= i3Step + 1;
		END_IF 
	
	34:
		IF u01.steam_header_flow > u01.SP_minimum_steam_bypass_flow_rate THEN
			i3Step														:= i3Step + 1;										// 13.a
		ELSE
			sError														:= gsSteamBypassMinFlowRateError;					// 13.b
			i3Step														:= 80;
		END_IF
	
	35:
		IF tonTimer.Q OR u01.purge_product_line_temp > u01.SP_steam_bypass_temperature THEN									// 14
			bTimer														:= FALSE;
			u01.steam_bypass_valve										:= FALSE;											// 15
			gsCycleStage												:= SEL(bAdsorptionActive, 'steam_bypass.wrap_up', 'steam_bypass.wrap_up.adsorption');	// 15.a
			u01.purge_product_pre_condenser_valve						:= FALSE;											// 16
			u01.product_vacuum_bypass_valve								:= FALSE;
			u01.product_condenser										:= FALSE;
			//u01.product_blower											:= FALSE;
			u.product_blower_vfd										:= 0;
			IF bAdsorptionActive THEN
				i3Step													:= 40;
			ELSE
				u01.steam_bypass_complete								:= TRUE;
				i3Step													:= 90;
			END_IF
		END_IF
		
		
//**** Complete Adsorption		
	40:
		IF tonAdsorptionTimer.Q THEN																						// 17.a.i
			bAdsorptionTimer											:= FALSE;
			P_M01_RS01.fan_vfd_percent									:= 0;												// 17.a.ii
			P_M01_RS02.fan_vfd_percent									:= 0;
			P_M01_RS03.fan_vfd_percent									:= 0;
			gsCycleStage												:= 'steam_bypass.wrap_up.turn_off_fans';			// 17.a.ii.1
			rTime														:= _FAN_RS_DELAY_TIME;
			i3Step														:= i3Step + 1;
		END_IF

	41:
		bTimer															:= TRUE;
		IF tonTimer.Q THEN
			bTimer														:= FALSE;
			P_M01_RS01.close_all_doors									:= TRUE;											// 17.a.iii
			P_M01_RS02.close_all_doors									:= TRUE;
			P_M01_RS03.close_all_doors									:= TRUE;
			gsCycleStage												:= 'steam_bypass.wrap_up.close_doors';				// 17.a.iii.1
			rTime														:= m01.SP_doorsopenclose_timedelay * _MINUTES;										// 17.a.iii.2
			i3Step														:= i3Step + 1;
		END_IF		

	42:
		bTimer															:= TRUE;
		bPass1															:= (P_M01.bRS01 AND P_M01_RS01.R_S.all_doors_closed) OR NOT P_M01.bRS01;		// 17.a.iii.3
		bPass2															:= (P_M01.bRS02 AND P_M01_RS02.R_S.all_doors_closed) OR NOT P_M01.bRS02;
		bPass3															:= (P_M01.bRS03 AND P_M01_RS03.R_S.all_doors_closed) OR NOT P_M01.bRS03;
		IF bPass1 AND bPass2 AND bPass3 THEN
			bTimer														:= FALSE;
			i3Step														:= i3Step + 1;
		ELSIF tonTimer.Q THEN
			bTimer														:= FALSE;
			sRS															:= SEL(NOT bPass1, SEL(NOT bPass2, _RS03, _RS02), _RS01);
			P_Alarms.M_Add_Alarm(F_Concat3(_U01, sRS, gsCycleStage), gsReactorDoorClosingError, gsSystemCannotRun);
			i3Step														:= i3Step + 1;
		END_IF
		
	43:
		P_M01_RS01.co2_sensors_off										:= TRUE;											// 17.a.iv
		P_M01_RS02.co2_sensors_off										:= TRUE;
		P_M01_RS03.co2_sensors_off										:= TRUE;
		bAdsorptionActive												:= FALSE;											// 17.a.v
		i3Step															:= 90;

	
//**** Process error		
	80:
		gsCycleStage													:= 'steam_bypass.error';
		sMessage														:= SEL(sMessage = gsRunWarmup, gsProcessCannotRun, sMessage);
		P_Alarms.M_Add_Alarm(CONCAT(_U01, gsCycleStage), sError, sMessage);
		i3Step															:= i3Step + 1;

//**** Stop process
	81:
		P_M01_RS01.co2_sensors_off										:= TRUE;
		P_M01_RS02.co2_sensors_off										:= TRUE;
		P_M01_RS03.co2_sensors_off										:= TRUE;
		P_M01_RS01.fan_vfd_percent										:= 0;
		P_M01_RS02.fan_vfd_percent										:= 0;
		P_M01_RS03.fan_vfd_percent										:= 0;
		rTime															:= _FAN_RS_DELAY_TIME;
		i3Step															:= i3Step + 1;

	82:
		bTimer															:= TRUE;
		IF tonTimer.Q THEN
			bTimer														:= FALSE;
			i3Step														:= i3Step + 1;
		END_IF

	83:
		//u01.product_blower												:= FALSE;
		u.product_blower_vfd											:= 0;
		u01.purge_product_pre_condenser_valve							:= FALSE;
		u01.product_vacuum_bypass_valve									:= FALSE;
		u01.product_vacuum_pump_vfd										:= 0;
		u01.product_vacuum_backfeed_valve								:= _CLOSED;
		u01.cooling_line_pre_condenser_valve							:= FALSE;
		u01.purge_product_pre_condenser_valve							:= FALSE;
		u01.product_vacuum_pump_vfd										:= u01.SP_product_vacuum_idle_vfd_percent;
		u01.product_vacuum_pump_isolation_valve							:= FALSE;
		u01.product_vacuum_outlet_isolation_valve						:= FALSE;
		u01.product_condenser											:= FALSE;
		rTime															:= _VALVE_TIME;
		i3Step															:= i3Step + 1;
		
	84:
		bTimer															:= TRUE;
		IF tonTimer.Q THEN
			bTimer														:= FALSE;
			i3Step														:= 90;
		END_IF
		
//**** Close process
	90:
		gsCycleStage													:= SEL(bComplete, 'steam_bypass.failed', 'steam_bypass.complete');
		bAdsorptionTimer												:= FALSE;
		u01.drainage_on													:= FALSE;
		rTime															:= _PROCESS_COMPLETE_TIME;
		i3Step															:= i3Step + 1;
		
	91:
		bTimer															:= TRUE;
		IF tonTimer.Q THEN
			bTimer														:= FALSE;
			gsCycleStage												:= '';
			i3Step														:= 0;
		END_IF
				
END_CASE

IF i3Step > 0 AND i3Step < 80 AND u01.shutdown_process THEN
	gsCycleStage														:= 'steam_bypass.stopping';
	i3Step																:= 81;
END_IF
END_ACTION

ACTION A8_Shutdown:
// Phase 0 - P_U01.A8_Shutdown
// Rev 1.0 - May 1, 2024

CASE i8Step OF

	0:	;

	1:	
		bComplete														:= FALSE;
		gsCycleStage													:= 'shutdown.initialize';							// 1.a
		u01.boiler_package												:= FALSE;											// 3
		i8Step															:= i8Step + 1;

	2:
		P_M01_RS01.fan_vfd_percent										:= 0;
		P_M01_RS02.fan_vfd_percent										:= 0;
		P_M01_RS03.fan_vfd_percent										:= 0;
		rTime															:= _PAUSE_TIME;
		i8Step															:= i8Step + 1;
		
	3:
		bTimer															:= TRUE;
		IF tonTimer.Q THEN
			bTimer														:= FALSE;						
			P_M01_RS01.close_all_doors									:= P_M01.bRS01;										// 4
			P_M01_RS02.close_all_doors									:= P_M01.bRS02;
			P_M01_RS03.close_all_doors									:= P_M01.bRS03;
			gsCycleStage												:= 'shutdown.close_doors';							// 4.a
			rTime														:= m01.SP_doorsopenclose_timedelay * _MINUTES;
			i8Step														:= i8Step + 1;
		END_IF

	4:
		bTimer															:= TRUE; 
		bPass1															:= (P_M01.bRS01 AND P_M01_RS01.R_S.all_doors_closed) OR NOT P_M01.bRS01;
		bPass2															:= (P_M01.bRS02 AND P_M01_RS02.R_S.all_doors_closed) OR NOT P_M01.bRS02;
		bPass3															:= (P_M01.bRS03 AND P_M01_RS03.R_S.all_doors_closed) OR NOT P_M01.bRS03;
		IF (bPass1 AND bPass2 AND bPass3) OR tonTimer.Q THEN
			IF tonTimer.Q THEN 
				sRS														:= SEL(NOT bPass1, SEL(NOT bPass2, _RS03, _RS02), _RS01);
				P_Alarms.M_Add_Alarm(F_Concat3(_U01, gsCycleStage, sRS), gsReactorDoorClosingError, gsSystemCannotRun);
			END_IF
			bTimer														:= FALSE;
			i8Step														:= i8Step + 1;
		END_IF

	5:
		P_M01_RS01.close_valves											:= P_M01.bRS01;										// 5		
		P_M01_RS02.close_valves											:= P_M01.bRS02;		
		P_M01_RS03.close_valves											:= P_M01.bRS03;
		gsCycleStage													:= 'shutdown.wrap_up';								// 5.a
		rTime															:= _VALVE_TIME;
		i8Step															:= i8Step + 1;
		
	6:
		bTimer															:= TRUE;
		IF tonTimer.Q THEN
			bTimer														:= FALSE;
			P_M01_RS01.co2_sensors_off									:= P_M01.bRS01;
			P_M01_RS02.co2_sensors_off									:= P_M01.bRS02;
			P_M01_RS03.co2_sensors_off									:= P_M01.bRS03;
			P_M01_RS01.close_repres_valves								:= P_M01.bRS01;
			P_M01_RS02.close_repres_valves								:= P_M01.bRS02;
			P_M01_RS03.close_repres_valves								:= P_M01.bRS03;
			i8Step														:= i8Step + 1;
		END_IF
		
	7:
		P_U01.bCloseXVValves											:= TRUE;
		u01.product_vacuum_backfeed_valve								:= 0;
		u01.product_vacuum_pump_vfd										:= 0;
		u01.product_condensate_pump										:= FALSE;
		u01.condensate_collection_tank_pump								:= FALSE;
		u01.product_condenser											:= FALSE;
		u01.dead_air_vacuum_pump										:= FALSE;
		//u01.product_blower												:= FALSE;
		u.product_blower_vfd											:= 0;
		rTime															:= _PAUSE_TIME;
		i8Step															:= i8Step + 1;

	8:
		bTimer															:= TRUE;
		bPass1															:= NOT M01_rs1.condensate_lsl;						// 6
		bPass2															:= NOT m01_rs2.condensate_lsl;
		bPass3															:= NOT m01_rs2.condensate_lsl;
		bPass4															:= NOT m01.condensate_from_cooling_and_purge_lines_lsl;
		bPass5															:= NOT u01.product_condensate_drum_lsh;
		bPass6															:= NOT u01.condensate_collection_tank_lsh;
		gsCycleStage													:= 'shutdown.drain';								// 6.a
		IF bPass1 AND bPass2 AND bPass3 AND bPass4 AND bPass5 AND bPass6 THEN
			bTimer														:= FALSE;
 		ELSIF tonTimer.Q THEN
			sError														:= SEL(NOT bPass1, '', F_concat3(_RS01, ' ', gsCondensateLslError));
			sError														:= SEL(NOT bPass2, sError, F_concat3(_RS02, ' ', gsCondensateLslError));
			sError														:= SEL(NOT bPass3, sError, F_concat3(_RS03, ' ', gsCondensateLslError));
			sError														:= SEL(NOT bPass4, sError, gsCondensateFromCoolingAndPurgeLinesLslError);
			sError														:= SEL(NOT bPass5, sError, gsProductCondensateDrumLshError);
			sError														:= SEL(NOT bPass6, sError, gsCondensateCollectionTankLshError);
			P_Alarms.M_Add_Alarm(_U01, sError, gsCheckOperation);
		END_IF
		i8Step															:= 90;
		
//**** Close process
	90:
		gsCycleStage													:= 'shutdown.complete';								// 7
		rTime															:= _PROCESS_COMPLETE_TIME;
		i8Step															:= i8Step + 1;
		
	91:
		bTimer															:= TRUE;
		IF tonTimer.Q THEN
			bTimer														:= FALSE;
			gsCycleStage												:= '';
			i8Step														:= 0;
		END_IF
				
END_CASE

IF i8Step > 0 AND i8Step < 80 AND u01.shutdown_process THEN
	gsCycleStage														:= 'shutdown.stopping';
	i8Step																:= 81;
END_IF
END_ACTION

ACTION A9_Pressure_Drop_Test:
// Phase 0 - P_U01.A9_Pressure_Drop_Test
// Rev 1.0 - June 3, 2024

CASE i9Step OF

	0:	;

	1:	
		bComplete														:= FALSE;
		gsCycleStage													:= 'pressure_drop_test.initialize';					// 3
		i9Step															:= i9Step + 1;

	2:	
		Ax_Process_Pre_Check();																								// 3.a																			
		IF bPreCheckDone THEN
			IF sError = '' THEN																								// 3.a.i
				u01.drainage_on											:= TRUE;											// 3.c
				u01.product_vacuum_pump_vfd								:= u01.SP_product_vacuum_idle_vfd_percent;			// 3d
				i9Step													:= i9Step + 1;
			ELSE
				sRS														:= '';
				sMessage												:= gsPressureDropTestCannotRun;						// 3.a.ii
				i9Step													:= 80;
			END_IF
		END_IF

	3:
		P_M01_RS01.open_repres_valves									:= P_M01.bRS01;										// 4
		P_M01_RS02.open_repres_valves									:= P_M01.bRS02;
		P_M01_RS03.open_repres_valves									:= P_M01.bRS03;
		rTime															:= _VALVE_TIME;
		i9Step															:= i9Step + 1;

	4:
		bTimer															:= TRUE;
		bPass1															:= (P_M01.bRS01 AND P_M01_RS01.repres_valves_clear) OR NOT P_M01.bRS01;
		bPass2															:= (P_M01.bRS02 AND P_M01_RS02.repres_valves_clear) OR NOT P_M01.bRS02;
		bPass3															:= (P_M01.bRS03 AND P_M01_RS03.repres_valves_clear) OR NOT P_M01.bRS03;
		IF bPass1 AND bPass2 AND bPass3 OR tonTimer.Q THEN
			bTimer														:= FALSE;
			i9Step														:= i9Step + 1;
		END_IF
		
	5:
		P_M01_RS01.open_all_doors										:= P_M01.bRS01;										// 5
		P_M01_RS02.open_all_doors										:= P_M01.bRS02;
		P_M01_RS03.open_all_doors										:= P_M01.bRS03;
		gsCycleStage													:= 'pressure_drop_test.open_doors';					// 5.a
		rTime															:= m01.SP_doorsopenclose_timedelay * _MINUTES;		// 5.b
		i9Step															:= i9Step + 1;

	6:
		bTimer															:= TRUE; 
		bPass1															:= (P_M01.bRS01 AND P_M01_RS01.R_S.all_doors_open) OR NOT P_M01.bRS01;	// 5.c
		bPass2															:= (P_M01.bRS02 AND P_M01_RS02.R_S.all_doors_open) OR NOT P_M01.bRS02;
		bPass3															:= (P_M01.bRS03 AND P_M01_RS03.R_S.all_doors_open) OR NOT P_M01.bRS03;
		IF bPass1 AND bPass2 AND bPass3 THEN
			bTimer														:= FALSE;
			iVfd_Speed													:= u01.SP_reactor_vfd_percent_step_size;			// 6
			bVfd_Speed_Up												:= TRUE;
			gsCycleStage												:= 'pressure_drop_test.pressure_drop_test';			// 6.a
			rTime														:= u01.SP_reactor_vfd_percent_step_duration * _MINUTES;	// 7
			i9Step														:= i9Step + 1;
		ELSIF tonTimer.Q THEN
			bTimer														:= FALSE;
			sRS															:= SEL(NOT bPass1, SEL(NOT bPass2, _RS03, _RS02), _RS01);
			sError														:= gsReactorDoorOpeningError;
			sMessage													:= gsPressureDropTestCannotRun;
			i9Step														:= 80;
		END_IF

	7:
		P_M01_RS01.fan_vfd_percent										:= SEL(P_M01.bRS01, 0, iVfd_Speed);
		P_M01_RS02.fan_vfd_percent										:= SEL(P_M01.bRS02, 0, iVfd_Speed);
		P_M01_RS03.fan_vfd_percent										:= SEL(P_M01.bRS03, 0, iVfd_Speed);
		i9Step															:= SEL(iVfd_Speed = 0, i9Step + 1, i9Step + 2);		//11

	8:
		bTimer															:= TRUE;
		IF tonTimer.Q THEN																									// 8
			bTimer														:= FALSE;
			IF bVfd_Speed_Up THEN
				IF iVfd_Speed + u01.SP_reactor_vfd_percent_step_size <= u01.SP_reactor_vfd_percent_maximum THEN
					iVfd_Speed											:= iVfd_Speed + u01.SP_reactor_vfd_percent_step_size;	// 9
				ELSE
					bVfd_Speed_Up										:= FALSE;
					iVfd_Speed											:= iVfd_Speed - u01.SP_reactor_vfd_percent_step_size;
				END_IF
			ELSE
				IF iVfd_Speed - u01.SP_reactor_vfd_percent_step_size >= 0 THEN
					iVfd_Speed											:= iVfd_Speed - u01.SP_reactor_vfd_percent_step_size;	// 10
				ELSE
					iVfd_Speed											:= 0;
				END_IF
			END_IF
			i9Step														:= i9Step - 1;
		END_IF

	9:
		bComplete														:= TRUE;
		gsCycleStage													:= 'pressure_drop_test.close_doors';				// 11.a
		P_M01_RS01.close_all_doors										:= P_M01.bRS01;										// 12
		P_M01_RS02.close_all_doors										:= P_M01.bRS02;
		P_M01_RS03.close_all_doors										:= P_M01.bRS03;
		rTime															:= m01.SP_doorsopenclose_timedelay * _MINUTES;										// 12.a
		i9Step															:= i9Step + 1;

	10:
		bTimer															:= TRUE;
		bPass1															:= (P_M01.bRS01 AND P_M01_RS01.R_S.all_doors_closed) OR NOT P_M01.bRS01;	// 12.b
		bPass2															:= (P_M01.bRS02 AND P_M01_RS02.R_S.all_doors_closed) OR NOT P_M01.bRS02;
		bPass3															:= (P_M01.bRS03 AND P_M01_RS03.R_S.all_doors_closed) OR NOT P_M01.bRS03;
		IF bPass1 AND bPass2 AND bPass3 THEN
			bTimer														:= FALSE;
			i9Step														:= i9Step + 1;
		ELSIF tonTimer.Q THEN
			bTimer														:= FALSE;
			sRS															:= SEL(NOT bPass1, SEL(NOT bPass2, _RS03, _RS02), _RS01);
			P_Alarms.M_Add_Alarm(F_Concat3(_U01, gsCycleStage, sRS), gsReactorDoorClosingError, gsUnableToCloseDoors);
			i9Step														:= 90;
		END_IF
		

//**** Process error		
	80:
		gsCycleStage													:= 'pressure_drop_test.error';
		P_Alarms.M_Add_Alarm(F_Concat3(_U01, sRS, gsCycleStage), sError, sMessage);
		i9Step															:= i9Step + 1;

//**** Stop process		
	81:
		u01.product_vacuum_pump_vfd										:= 0;
		P_M01_RS01.fan_vfd_percent										:= 0;
		//P_M01_RS02.fan_vfd_percent										:= 0;
		//P_M01_RS03.fan_vfd_percent										:= 0;
		i9Step															:= 90;
		
//**** Close process
	90:
		gsCycleStage													:= SEL(bComplete, 'pressure_drop_test.failed', 'pressure_drop_test.complete');	// 13
		u01.drainage_on													:= FALSE;
		rTime															:= _PROCESS_COMPLETE_TIME;
		i9Step															:= i9Step + 1;
		
	91:
		bTimer															:= TRUE;
		IF tonTimer.Q THEN
			bTimer														:= FALSE;
			gsCycleStage												:= '';
			i9Step														:= 0;
		END_IF
				
END_CASE

IF i9Step > 0 AND i9Step < 80 AND u01.shutdown_process THEN
	gsCycleStage														:= 'pressure_drop_test.stopping';
	i9Step																:= 81;
END_IF
END_ACTION

ACTION Ax_Process_Pre_Check:
// Phase 0 - P_U01.Ax_Process_Pre_Check
// Rev 1.0 - April 30, 2024

CASE iAxStep OF

	0:	;

	1:	
		sError															:= '';
		bPreCheckDone													:= FALSE;
		P_M01_RS01.close_valves											:= P_M01.bRS01;
		P_M01_RS02.close_valves											:= P_M01.bRS02;
		P_M01_RS03.close_valves											:= P_M01.bRS03;
		P_M01_RS01.retract_all_clamps									:= P_M01.bRS01;
		P_M01_RS02.retract_all_clamps									:= P_M01.bRS02;
		P_M01_RS03.retract_all_clamps									:= P_M01.bRS03;
		rTime															:= _VALVE_TIME;
		iAxStep															:= iAxStep + 1;
	
	2:	
		bTimer															:= TRUE;
		bPass1															:= (P_M01.bRS01 AND P_M01_RS01.R_S.valves_clear AND m01_rs1.steam_control_valve_position < _VALVE_CLOSED) OR NOT P_M01.bRS01;
		bPass2															:= (P_M01.bRS02 AND P_M01_RS02.R_S.valves_clear AND m01_rs2.steam_control_valve_position < _VALVE_CLOSED) OR NOT P_M01.bRS02;
		bPass3															:= (P_M01.bRS03 AND P_M01_RS03.R_S.valves_clear AND m01_rs3.steam_control_valve_position < _VALVE_CLOSED) OR NOT P_M01.bRS03;
		IF bPass1 AND bPass2 AND bPass3 THEN
			bTimer														:= FALSE;
			iAxStep														:= iAxStep + 1;
		ELSIF tonTimer.Q THEN
			sError														:= 'Valve Error';
			iAxStep														:= 99;
		END_IF

	3:
		IF (P_M01_RS01.inlet_air_high_temp_count + P_M01_RS02.inlet_air_high_temp_count + P_M01_RS03.inlet_air_high_temp_count) <= _HIGH_CART_READINGS_MAX THEN
			iAxStep														:= iAxStep + 1;
		ELSE
			sError														:= gsHighTempCountError;
			iAxStep														:= 99;
		END_IF

	4:
		bPass1															:= (P_M01.bRS01 AND P_M01_RS01.R_S.all_clamps_retracted) OR NOT P_M01.bRS01; 
		bPass2															:= (P_M01.bRS02 AND P_M01_RS02.R_S.all_clamps_retracted) OR NOT P_M01.bRS02; 
		bPass3															:= (P_M01.bRS03 AND P_M01_RS03.R_S.all_clamps_retracted) OR NOT P_M01.bRS03; 
		IF bPass1 AND bPass2 AND bPass3 THEN
			iAxStep														:= iAxStep + 1;
		ELSE
			sError														:= gsClampRetractError;
			iAxStep														:= 99;
		END_IF
		
	5:
		IF NOT u.os_air_unsafe_temp THEN
			iAxStep														:= iAxStep + 1;
		ELSE
			sError														:= gsInletAirTempRangeError;
			iAxStep														:= 99;
		END_IF
		
	6:
		bPass1															:= (P_M01.bRS01 AND P_M01_RS01.average_pressure_within_ambient) OR NOT P_M01.bRS01;
		bPass2															:= (P_M01.bRS02 AND P_M01_RS02.average_pressure_within_ambient) OR NOT P_M01.bRS02;
		bPass3															:= (P_M01.bRS03 AND P_M01_RS03.average_pressure_within_ambient) OR NOT P_M01.bRS03;
		IF NOT bPass1 OR NOT bPass2 OR NOT bPass3 THEN
			sError														:=  gsAmbientPressureError;
		END_IF
		iAxStep															:= 99;
		
	99:
		bTimer															:= FALSE;
		bPreCheckDone													:= TRUE;
		iAxStep															:= 0;
				
END_CASE
END_ACTION

METHOD M_Repres_Valve_Error : STRING
VAR_INPUT
END_VAR
VAR
	sErr																: STRING	:= '';
END_VAR
// Phase 0 - P_U01.M_Repres_Valve_Error
// Rev 1.0 - March 12, 2024

IF P_M01.bRS03 THEN
	;//sErr																:= SEL(P_M01_RS03_R4.bRepresValveClear, CONCAT(_RS03, _R4), sErr);
	//sErr																:= SEL(P_M01_RS03_R3.bRepresValveClear, CONCAT(_RS03, _R3), sErr);
	//sErr																:= SEL(P_M01_RS03_R2.bRepresValveClear, CONCAT(_RS03, _R2), sErr);
	//sErr																:= SEL(P_M01_RS03_R1.bRepresValveClear, CONCAT(_RS03, _R1), sErr);
END_IF                                                                                                                                   
IF P_M01.bRS02 THEN                                                                                                                       
	;//sErr																:= SEL(P_M01_RS02_R4.bRepresValveClear, CONCAT(_RS02, _R4), sErr);
	//sErr																:= SEL(P_M01_RS02_R3.bRepresValveClear, CONCAT(_RS02, _R3), sErr);
	//sErr																:= SEL(P_M01_RS02_R2.bRepresValveClear, CONCAT(_RS02, _R2), sErr);
	//sErr																:= SEL(P_M01_RS02_R1.bRepresValveClear, CONCAT(_RS02, _R1), sErr);
END_IF                                                                                                                                   
IF P_M01.bRS01 THEN                                                                                                                       
	//sErr																:= SEL(P_M01_RS01_R4.bRepresValveClear, CONCAT(_RS01, _R4), sErr);
	//sErr																:= SEL(P_M01_RS01_R3.bRepresValveClear, CONCAT(_RS01, _R3), sErr);
	//sErr																:= SEL(P_M01_RS01_R2.bRepresValveClear, CONCAT(_RS01, _R2), sErr);
	//sErr																:= SEL(P_M01_RS01.repres_valves_clear, CONCAT(_RS01, _R1), sErr);
END_IF
M_Repres_Valve_Error													:= SEL(sErr <> '', sErr, CONCAT(sErr, gsRepressurizationValveError));
END_METHOD

END_PROGRAM

// ---- POUs/Function_Blocks/FB_Digital_Out.TcPOU
FUNCTION_BLOCK FB_Digital_Out
VAR_OUTPUT
	Output																: BOOL;
END_VAR
VAR_IN_OUT
	Input1																: BOOL;
	Input2																: BOOL;
END_VAR
VAR
	blast1																: BOOL;
	blast2																: BOOL;
END_VAR

// Phase 0 - FB_Digital_Out
// Rev 1.0 - March 29, 2024

// Allows two inputs (HMI/Utility vs Reactor Set) to control one point. Output mirrors the last input (On or Off) and both inputs are changed to the new value.

IF Input1 <> bLast1 THEN
	bLast1																:= Input1;
	Input2																:= Input1;
	bLast2																:= Input1;
ELSIF Input2 <> bLast2 THEN
	bLast2																:= Input2;
	Input1																:= Input2;
	bLast1																:= Input2;
END_IF
Output																	:= Input1;

END_FUNCTION_BLOCK

// ---- POUs/Function_Blocks/FB_Analog_Out.TcPOU
FUNCTION_BLOCK FB_Analog_Out
VAR_INPUT
END_VAR
VAR_IN_OUT
	Input1																: REAL;
	Input2																: REAL;
END_VAR
VAR
	Last1																: REAL;
	Last2																: REAL;
END_VAR

// Phase 0 - FB_Analog_Out
// Rev 1.0 - April 3, 2024

IF Input2 <> Last2 THEN
	Last2																:= Input2;
	Input1																:= Input2;
	Last1																:= Input2;
ELSIF Input1 <> Last1 THEN
	Last1																:= Input1;
	Input2																:= Input1;
	Last2																:= Input1;
END_IF

END_FUNCTION_BLOCK

// ---- POUs/Function_Blocks/FB_Integer_Out.TcPOU
FUNCTION_BLOCK FB_Integer_Out
VAR_INPUT
END_VAR
VAR_IN_OUT
	Input1																: INT;
	Input2																: INT;
END_VAR
VAR
	Last1																: INT;
	Last2																: INT;
END_VAR

// Phase 0 - FB_Integer_Out
// Rev 1.0 - April 24, 2024

IF Input2 <> Last2 THEN
	Last2																:= Input2;
	Input1																:= Input2;
	Last1																:= Input2;
ELSIF Input1 <> Last1 THEN
	Last1																:= Input1;
	Input2																:= Input1;
	Last2																:= Input1;
END_IF

END_FUNCTION_BLOCK

// ---- POUs/Function_Blocks/FB_Vacuum_Pump.TcPOU
FUNCTION_BLOCK FB_Vacuum_Pump
VAR_IN_OUT
	Pump_Reset															: BOOL;
END_VAR
VAR_INPUT
	Enable																: BOOL;
	Purge_Time															: REAL;
	Safety1																: BOOL;
	Safety2																: BOOL;
	Safety3																: BOOL;
END_VAR
VAR_OUTPUT
	Error																: INT;
	Pump_On																: BOOL;
	Seal_Purge_Valve													: BOOL;
	Purge_Solenoid_Valve												: BOOL;
END_VAR
VAR
	bErrorOn															: BOOL;
	bError1																: BOOL;
	bError2																: BOOL;
	bError3																: BOOL;
	bStop																: BOOL;
	tonPurge															: TON;
	rtrigError															: R_TRIG;
END_VAR

// Phase 0 - FB_Vacuum_Pump
// Rev 1.0 - April 17, 2024

Error																	:= 0;
bError1																	:= NOT Safety1;
bError2																	:= NOT Safety2;
bError3																	:= NOT Safety3;

rtrigError(CLK:= bError1 OR bError2 OR bError3);
IF rtrigError.Q THEN
	bErrorOn															:= TRUE;
	bStop																:= FALSE;
	Pump_On																:= FALSE;
	Seal_Purge_Valve													:= FALSE;
	Purge_Solenoid_Valve												:= FALSE;
	u01.product_vacuum_pump_isolation_valve								:= FALSE;
	u01.product_vacuum_pump_vfd											:= 0;
	Error																:= SEL(bError1, SEL(bError2, SEL(bError3, 0, 3), 2), 1);
END_IF

IF NOT bErrorOn THEN
	IF tonPurge.Q THEN
		bStop															:= FALSE;
		Pump_On															:= FALSE;
		Purge_Solenoid_Valve											:= FALSE;
		Seal_Purge_Valve												:= FALSE;
		u01.product_vacuum_pump_vfd										:= 0;
	ELSIF Enable AND NOT Pump_On THEN
		Pump_On															:= TRUE;
		Seal_Purge_Valve												:= TRUE;
		u01.product_vacuum_pump_isolation_valve							:= TRUE;
		u01.product_vacuum_pump_vfd										:= u01.SP_product_vacuum_idle_vfd_percent;
	ELSIF NOT Enable AND Pump_On AND NOT bStop THEN
		bStop															:= TRUE;
		Purge_Solenoid_Valve											:= TRUE;
		u01.product_vacuum_pump_isolation_valve							:= FALSE;
		u01.product_vacuum_pump_vfd										:= u01.SP_product_vacuum_purge_vfd_percent;
	END_IF
END_IF

tonPurge(IN:= bStop, PT:= REAL_TO_TIME(Purge_Time * _MINUTES));

IF Pump_Reset OR NOT Enable THEN
	bErrorOn															:= FALSE;
	Pump_Reset															:= FALSE;
END_IF

END_FUNCTION_BLOCK

// ---- POUs/Reactor_Set_01/P_M01_RS01.TcPOU
PROGRAM P_M01_RS01
VAR_INPUT
	stop_rs_automode													: BOOL;
	clear_rs_pause														: BOOL;
	close_valves														: BOOL;
	close_all_doors														: BOOL;
	open_all_doors														: BOOL;
	retract_all_clamps													: BOOL;
	extend_all_clamps													: BOOL;
	open_repres_valves													: BOOL;
	close_repres_valves													: BOOL;
	co2_sensors_off														: BOOL;
	co2_inside_sensors_on												: BOOL;
	co2_outside_sensors_on												: BOOL;
	fan_vfd_percent														: REAL		:= 0;
END_VAR
VAR_OUTPUT
	repres_valves_clear													: BOOL;
	average_pressure_within_ambient										: BOOL;
	reactor_done														: BOOL;
	utility_error														: BOOL;
	cancel_reactor_set													: BOOL;
	cancel_all_reactor_sets												: BOOL;
	inlet_air_high_temp_count											: INT;
	open_inlet_doors													: BOOL;
	open_outlet_doors													: BOOL;
	close_inlet_doors													: BOOL;
	close_outlet_doors													: BOOL;
	open_doors															: BOOL;
	close_doors															: BOOL;
	inlet_door_clamps_extend											: BOOL;
	outlet_door_clamps_extend											: BOOL;
	inlet_door_clamps_retract											: BOOL;
	outlet_door_clamps_retract											: BOOL;
	extend_clamps														: BOOL;
	retract_clamps														: BOOL;
END_VAR
VAR
	R_S																	: Reactor_Set;

	fb_RS																: FB_Reactor_Set();
	fb_RS_IO															: FB_Reactor_Set_IO();
	fb_R1_IO															: FB_Reactor_IO();
	fb_R2_IO															: FB_Reactor_IO();
	fb_R3_IO															: FB_Reactor_IO();
	fb_R4_IO															: FB_Reactor_IO();
	
	fb_Fan_Vfd															: FB_Analog_Out();
	
	rAveragePressure													: REAL;
	rValve																: REAL;
	rPos																: REAL;
	rFanOldVfdPercent													: REAL		:= 0;
	
	iCount																: INT;
	iVacuumStatus														: INT;
	iError																: INT;
	
	bR1OverMaxPressure													: BOOL;
	bR2OverMaxPressure													: BOOL;
	bR3OverMaxPressure													: BOOL;
	bR4OverMaxPressure													: BOOL;
	
	bR1InletCO2Error													: BOOL;
	bR1InletH2OError													: BOOL;
	bR1OutletCO2Error													: BOOL;
	bR1OutletH2OError													: BOOL;
	bR1AirFlowError														: BOOL;
	bR1FilterDiffPresError												: BOOL;
	bR1SorbentDiffPresError												: BOOL;
	bR1FanDiffPresError													: BOOL;
	bR1ReactorPresError													: BOOL;
	
	bR2InletCO2Error													: BOOL;
	bR2InletH2OError													: BOOL;
	bR2OutletCO2Error													: BOOL;
	bR2OutletH2OError													: BOOL;
	bR2AirFlowError														: BOOL;
	bR2FilterDiffPresError												: BOOL;
	bR2SorbentDiffPresError												: BOOL;
	bR2FanDiffPresError													: BOOL;
	bR2ReactorPresError													: BOOL;
	
	bR3InletCO2Error													: BOOL;
	bR3InletH2OError													: BOOL;
	bR3OutletCO2Error													: BOOL;
	bR3OutletH2OError													: BOOL;
	bR3AirFlowError														: BOOL;
	bR3FilterDiffPresError												: BOOL;
	bR3SorbentDiffPresError												: BOOL;
	bR3FanDiffPresError													: BOOL;
	bR3ReactorPresError													: BOOL;
	
	bR4InletCO2Error													: BOOL;
	bR4InletH2OError													: BOOL;
	bR4OutletCO2Error													: BOOL;
	bR4OutletH2OError													: BOOL;
	bR4AirFlowError														: BOOL;
	bR4FilterDiffPresError												: BOOL;
	bR4SorbentDiffPresError												: BOOL;
	bR4FanDiffPresError													: BOOL;
	bR4ReactorPresError													: BOOL;
	
	stop_reactor_set													: BOOL;
	clear_reactor_set_pause												: BOOL;
END_VAR

// Phase 0 - P_M01_RS01
// Rev 1.0 - May 11, 2024

giEvacuationErrorRS														:= SEL(giEvacuationErrorRS = 1, giEvacuationErrorRS, 0);
giDesorptionErrorRS														:= SEL(giDesorptionErrorRS = 1, giDesorptionErrorRS, 0);
giSafeShutdown1RS														:= SEL(giSafeShutdown1RS = 1, giSafeShutdown1RS, 0);
giSafeShutdown23RS														:= SEL(giSafeShutdown23RS = 1, giSafeShutdown23RS, 0);

stop_reactor_set														:= stop_rs_automode;
stop_rs_automode														:= FALSE;
clear_reactor_set_pause													:= clear_rs_pause;
clear_rs_pause															:= FALSE;

A_Reactor_Set();

// REACTOR OUTPUTS
IF open_repres_valves OR R_S.open_repres_valves THEN
	fb_R1_IO.bRepresValve												:= TRUE;
	fb_R2_IO.bRepresValve												:= TRUE;
	fb_R3_IO.bRepresValve												:= TRUE;
	fb_R4_IO.bRepresValve												:= TRUE;
	open_repres_valves													:= FALSE;
END_IF
IF close_repres_valves OR R_S.close_repres_valves THEN
	fb_R1_IO.bRepresValve												:= FALSE;
	fb_R2_IO.bRepresValve												:= FALSE;
	fb_R3_IO.bRepresValve												:= FALSE;
	fb_R4_IO.bRepresValve												:= FALSE;
	close_repres_valves													:= FALSE;
END_IF

repres_valves_clear														:= fb_R1_IO.repres_valve_clear AND fb_R2_IO.repres_valve_clear AND fb_R3_IO.repres_valve_clear AND fb_R4_IO.repres_valve_clear;
IF NOT repres_valves_clear THEN
	R_S.repres_valve_error												:= SEL(fb_R4_IO.repres_valve_clear, CONCAT(_R4, gsRepressurizationValveError), '');
	R_S.repres_valve_error												:= SEL(fb_R3_IO.repres_valve_clear, CONCAT(_R3, gsRepressurizationValveError), R_S.repres_valve_error);
	R_S.repres_valve_error												:= SEL(fb_R2_IO.repres_valve_clear, CONCAT(_R2, gsRepressurizationValveError), R_S.repres_valve_error);
	R_S.repres_valve_error												:= SEL(fb_R1_IO.repres_valve_clear, CONCAT(_R1, gsRepressurizationValveError), R_S.repres_valve_error);
ELSE
	R_S.repres_valve_error												:= '';
END_IF

fb_Fan_Vfd(Input1:= fan_vfd_percent, Input2:= R_S.fan_vfd_percent);
IF fan_vfd_percent <> rFanOldVfdPercent THEN
	fb_R1_IO.fan_vfd_input											:= fan_vfd_percent;
	fb_R2_IO.fan_vfd_input											:= fan_vfd_percent;
	fb_R3_IO.fan_vfd_input											:= fan_vfd_percent;
	fb_R4_IO.fan_vfd_input											:= fan_vfd_percent;
	rFanOldVfdPercent													:= fan_vfd_percent;
END_IF
		
A_Reactor1_IO();
A_Reactor2_IO();
A_Reactor3_IO();
A_Reactor4_IO();

inlet_air_high_temp_count												:= fb_R1_IO.adsorption_high_temp_count + fb_R2_IO.adsorption_high_temp_count + fb_R3_IO.adsorption_high_temp_count + fb_R4_IO.adsorption_high_temp_count;
R_S.inlet_air_high_temp_count											:= inlet_air_high_temp_count;
R_S.desorption_high_temp_count											:= fb_R1_IO.desorption_high_temp_count + fb_R2_IO.desorption_high_temp_count + fb_R3_IO.desorption_high_temp_count + fb_R4_IO.desorption_high_temp_count;
R_S.vacuum_cooling_high_temp_count										:= fb_R1_IO.vacuum_cooling_high_temp_count + fb_R2_IO.vacuum_cooling_high_temp_count + fb_R3_IO.vacuum_cooling_high_temp_count + fb_R4_IO.vacuum_cooling_high_temp_count;
R_S.sorbent_high_temp													:= F_HighestReal(fb_R1_IO.sorbent_high_temp, fb_R2_IO.sorbent_high_temp, fb_R3_IO.sorbent_high_temp, fb_R4_IO.sorbent_high_temp);

m01_rs1_r1.reactor_wall_temp											:= F_Temperature(m01_rs1_r1.TT_05, m01_rs1_r1.reactor_wall_temp_offset);
m01_rs1_r1.outlet_line_temp												:= F_Temperature(m01_rs1_r1.TT_06, m01_rs1_r1.outlet_line_temp_offset);
m01_rs1_r2.reactor_wall_temp											:= F_Temperature(m01_rs1_r2.TT_05, m01_rs1_r2.reactor_wall_temp_offset);
m01_rs1_r2.outlet_line_temp												:= F_Temperature(m01_rs1_r2.TT_06, m01_rs1_r2.outlet_line_temp_offset);
m01_rs1_r3.reactor_wall_temp											:= F_Temperature(m01_rs1_r3.TT_05, m01_rs1_r3.reactor_wall_temp_offset);
m01_rs1_r3.outlet_line_temp												:= F_Temperature(m01_rs1_r3.TT_06, m01_rs1_r3.outlet_line_temp_offset);
m01_rs1_r4.reactor_wall_temp											:= F_Temperature(m01_rs1_r4.TT_05, m01_rs1_r4.reactor_wall_temp_offset);
m01_rs1_r4.outlet_line_temp												:= F_Temperature(m01_rs1_r4.TT_06, m01_rs1_r4.outlet_line_temp_offset);


// CO2 SENSOR HANDLING
IF co2_sensors_off OR R_S.co2_sensors_off THEN
	fb_R1_IO.co2_sensor_config											:= 0;
	fb_R2_IO.co2_sensor_config											:= 0;
	fb_R3_IO.co2_sensor_config											:= 0;
	fb_R4_IO.co2_sensor_config											:= 0;
	co2_sensors_off														:= FALSE;
ELSIF co2_inside_sensors_on OR R_S.co2_inside_sensors_on THEN
	fb_R1_IO.co2_sensor_config											:= 1;
	fb_R2_IO.co2_sensor_config											:= 1;
	fb_R3_IO.co2_sensor_config											:= 1;
	fb_R4_IO.co2_sensor_config											:= 1;
	co2_inside_sensors_on												:= FALSE;
ELSIF co2_outside_sensors_on OR R_S.co2_outside_sensors_on THEN
	fb_R1_IO.co2_sensor_config											:= 2;
	fb_R2_IO.co2_sensor_config											:= 2;
	fb_R3_IO.co2_sensor_config											:= 2;
	fb_R4_IO.co2_sensor_config											:= 2;
	co2_outside_sensors_on												:= FALSE;
END_IF
 
// DOORS & CLAMPS
inlet_door_clamps_extend												:= FALSE;	
outlet_door_clamps_extend												:= FALSE;
inlet_door_clamps_retract												:= FALSE;	
outlet_door_clamps_retract												:= FALSE;
extend_clamps															:= FALSE;
retract_clamps															:= FALSE;
IF extend_all_clamps OR R_S.extend_all_clamps THEN
	extend_clamps														:= TRUE;
	extend_all_clamps													:= FALSE;
END_IF
IF retract_all_clamps OR R_S.retract_all_clamps THEN
	retract_clamps														:= TRUE;	
	retract_all_clamps													:= FALSE;
END_IF
R_S.all_clamps_extended													:= fb_R1_IO.door_clamps_extended AND fb_R2_IO.door_clamps_extended AND fb_R3_IO.door_clamps_extended AND fb_R4_IO.door_clamps_extended; 
R_S.all_clamps_retracted												:= fb_R1_IO.door_clamps_retracted AND fb_R2_IO.door_clamps_retracted AND fb_R3_IO.door_clamps_retracted AND fb_R4_IO.door_clamps_retracted;

open_inlet_doors														:= FALSE;
open_outlet_doors														:= FALSE;
close_inlet_doors														:= FALSE;
close_outlet_doors														:= FALSE;
open_doors																:= FALSE;
close_doors																:= FALSE;
IF open_all_doors OR R_S.open_all_doors THEN
	open_doors															:= TRUE;
	open_all_doors														:= FALSE;
END_IF
fb_R1_IO.close_doors													:= FALSE;
IF close_all_doors OR R_S.close_all_doors THEN
	close_doors															:= TRUE;
	close_all_doors														:= FALSE;
END_IF
R_S.all_doors_open														:= fb_R1_IO.doors_open AND fb_R2_IO.doors_open AND fb_R3_IO.doors_open AND fb_R4_IO.doors_open;
R_S.all_doors_closed													:= fb_R1_IO.doors_closed AND fb_R2_IO.doors_closed AND fb_R3_IO.doors_closed AND fb_R4_IO.doors_closed;

m01_rs1_r1.inlet_co2													:= F_AnalogIn(m01_rs1_r1.AT_01, m01_rs1_r1.inlet_co2_low, m01_rs1_r1.inlet_co2_high, m01_rs1_r1.inlet_co2_min, m01_rs1_r1.inlet_co2_offset);
bR1InletCO2Error														:= P_Alarms.M_Check_Error(m01_rs1_r1.inlet_co2_error, bR1InletCO2Error, CONCAT(_RS01, _R1), gsInletCO2SensorError, gsProcessWillContinue);
m01_rs1_r1.inlet_h2o													:= F_AnalogIn(m01_rs1_r1.AT_02, m01_rs1_r1.inlet_h2o_low, m01_rs1_r1.inlet_h2o_high, m01_rs1_r1.inlet_h2o_min, m01_rs1_r1.inlet_h2o_offset);
bR1InletH2OError														:= P_Alarms.M_Check_Error(m01_rs1_r1.inlet_h2o_error, bR1InletH2OError, CONCAT(_RS01, _R1), gsInletH2OSensorError, gsProcessWillContinue);
m01_rs1_r1.outlet_co2													:= F_AnalogIn(m01_rs1_r1.AT_03, m01_rs1_r1.outlet_co2_low, m01_rs1_r1.outlet_co2_high, m01_rs1_r1.outlet_co2_min, m01_rs1_r1.outlet_co2_offset);
bR1OutletCO2Error														:= P_Alarms.M_Check_Error(m01_rs1_r1.outlet_co2_error, bR1OutletCO2Error, CONCAT(_RS01, _R1), gsOutletCO2SensorError, gsProcessWillContinue);
m01_rs1_r1.outlet_h2o													:= F_AnalogIn(m01_rs1_r1.AT_04, m01_rs1_r1.outlet_h2o_low, m01_rs1_r1.outlet_h2o_high, m01_rs1_r1.outlet_h2o_min, m01_rs1_r1.outlet_h2o_offset);
bR1OutletH2OError														:= P_Alarms.M_Check_Error(m01_rs1_r1.outlet_h2o_error, bR1OutletH2OError, CONCAT(_RS01, _R1), gsOutletH2OSensorError, gsProcessWillContinue);
m01_rs1_r1.air_flow														:= F_AnalogIn(m01_rs1_r1.FT_01, m01_rs1_r1.air_flow_low, m01_rs1_r1.air_flow_high, m01_rs1_r1.air_flow_min, m01_rs1_r1.air_flow_offset);
bR1AirFlowError															:= P_Alarms.M_Check_Error(m01_rs1_r1.air_flow_error, bR1AirFlowError, CONCAT(_RS01, _R1), gsAirFlowSensorError, gsProcessWillContinue);
m01_rs1_r1.filter_diff_pres												:= F_AnalogIn(m01_rs1_r1.PDT_01, m01_rs1_r1.filter_diff_pres_low, m01_rs1_r1.filter_diff_pres_high, m01_rs1_r1.filter_diff_pres_min, m01_rs1_r1.filter_diff_pres_offset);
bR1FilterDiffPresError													:= P_Alarms.M_Check_Error(m01_rs1_r1.filter_diff_pres_error, bR1FilterDiffPresError, CONCAT(_RS01, _R1), gsFilterDiffPresSensorError, gsProcessWillContinue);
m01_rs1_r1.sorbent_diff_pres											:= F_AnalogIn(m01_rs1_r1.PDT_02, m01_rs1_r1.sorbent_diff_pres_low, m01_rs1_r1.sorbent_diff_pres_high, m01_rs1_r1.sorbent_diff_pres_min, m01_rs1_r1.sorbent_diff_pres_offset,);
bR1SorbentDiffPresError													:= P_Alarms.M_Check_Error(m01_rs1_r1.sorbent_diff_pres_error, bR1SorbentDiffPresError, CONCAT(_RS01, _R1), gsSorbentDiffPresSensorError, gsProcessWillContinue);
m01_rs1_r1.fan_diff_pres												:= F_AnalogIn(m01_rs1_r1.PDT_03, m01_rs1_r1.fan_diff_pres_low, m01_rs1_r1.fan_diff_pres_high, m01_rs1_r1.fan_diff_pres_min, m01_rs1_r1.fan_diff_pres_offset);
bR1FanDiffPresError														:= P_Alarms.M_Check_Error(m01_rs1_r1.fan_diff_pres_error, bR1FanDiffPresError, CONCAT(_RS01, _R1), gsFanDiffPresSensorError, gsProcessWillContinue);
m01_rs1_r1.reactor_pres													:= F_AnalogIn(m01_rs1_r1.PT_01, m01_rs1_r1.reactor_pres_low, m01_rs1_r1.reactor_pres_high, m01_rs1_r1.reactor_pres_min, m01_rs1_r1.reactor_pres_offset);
bR1ReactorPresError														:= P_Alarms.M_Check_Error(m01_rs1_r1.reactor_pres_error, bR1ReactorPresError, CONCAT(_RS01, _R1), gsReactorPresSensorError, gsProcessWillContinue);
R_S.R1_reactor_pres														:= m01_rs1_r1.reactor_pres;
R_S.R1_reactor_pres_error												:= bR1ReactorPresError;
bR1OverMaxPressure														:= NOT m01_rs1_r1.reactor_pres_error AND m01_rs1_r1.reactor_pres > m01.SP_maximum_safe_reactor_steam_pressure;

m01_rs1_r2.inlet_co2													:= F_AnalogIn(m01_rs1_r2.AT_01, m01_rs1_r2.inlet_co2_low, m01_rs1_r2.inlet_co2_high, m01_rs1_r2.inlet_co2_min, m01_rs1_r2.inlet_co2_offset);
bR2InletCO2Error														:= P_Alarms.M_Check_Error(m01_rs1_r2.inlet_co2_error, bR2InletCO2Error, CONCAT(_RS01, _R2), gsInletCO2SensorError, gsProcessWillContinue);
m01_rs1_r2.inlet_h2o													:= F_AnalogIn(m01_rs1_r2.AT_02, m01_rs1_r2.inlet_h2o_low, m01_rs1_r2.inlet_h2o_high, m01_rs1_r2.inlet_h2o_min, m01_rs1_r2.inlet_h2o_offset);
bR2InletH2OError														:= P_Alarms.M_Check_Error(m01_rs1_r2.inlet_h2o_error, bR2InletH2OError, CONCAT(_RS01, _R2), gsInletH2OSensorError, gsProcessWillContinue);
m01_rs1_r2.outlet_co2													:= F_AnalogIn(m01_rs1_r2.AT_03, m01_rs1_r2.outlet_co2_low, m01_rs1_r2.outlet_co2_high, m01_rs1_r2.outlet_co2_min, m01_rs1_r2.outlet_co2_offset);
bR2OutletCO2Error														:= P_Alarms.M_Check_Error(m01_rs1_r2.outlet_co2_error, bR2OutletCO2Error, CONCAT(_RS01, _R2), gsOutletCO2SensorError, gsProcessWillContinue);
m01_rs1_r2.outlet_h2o													:= F_AnalogIn(m01_rs1_r2.AT_04, m01_rs1_r2.outlet_h2o_low, m01_rs1_r2.outlet_h2o_high, m01_rs1_r2.outlet_h2o_min, m01_rs1_r2.outlet_h2o_offset);
bR2OutletH2OError														:= P_Alarms.M_Check_Error(m01_rs1_r2.outlet_h2o_error, bR2OutletH2OError, CONCAT(_RS01, _R2), gsOutletH2OSensorError, gsProcessWillContinue);
m01_rs1_r2.air_flow														:= F_AnalogIn(m01_rs1_r2.FT_01, m01_rs1_r2.air_flow_low, m01_rs1_r2.air_flow_high, m01_rs1_r2.air_flow_min, m01_rs1_r2.air_flow_offset);
bR2AirFlowError															:= P_Alarms.M_Check_Error(m01_rs1_r2.air_flow_error, bR2AirFlowError, CONCAT(_RS01, _R2), gsAirFlowSensorError, gsProcessWillContinue);
m01_rs1_r2.filter_diff_pres												:= F_AnalogIn(m01_rs1_r2.PDT_01, m01_rs1_r2.filter_diff_pres_low, m01_rs1_r2.filter_diff_pres_high, m01_rs1_r2.filter_diff_pres_min, m01_rs1_r2.filter_diff_pres_offset);
bR2FilterDiffPresError													:= P_Alarms.M_Check_Error(m01_rs1_r2.filter_diff_pres_error, bR2FilterDiffPresError, CONCAT(_RS01, _R2), gsFilterDiffPresSensorError, gsProcessWillContinue);
m01_rs1_r2.sorbent_diff_pres											:= F_AnalogIn(m01_rs1_r2.PDT_02, m01_rs1_r2.sorbent_diff_pres_low, m01_rs1_r2.sorbent_diff_pres_high, m01_rs1_r2.sorbent_diff_pres_min, m01_rs1_r2.sorbent_diff_pres_offset,);
bR2SorbentDiffPresError													:= P_Alarms.M_Check_Error(m01_rs1_r2.sorbent_diff_pres_error, bR2SorbentDiffPresError, CONCAT(_RS01, _R2), gsSorbentDiffPresSensorError, gsProcessWillContinue);
m01_rs1_r2.fan_diff_pres												:= F_AnalogIn(m01_rs1_r2.PDT_03, m01_rs1_r2.fan_diff_pres_low, m01_rs1_r2.fan_diff_pres_high, m01_rs1_r2.fan_diff_pres_min, m01_rs1_r2.fan_diff_pres_offset);
bR2FanDiffPresError														:= P_Alarms.M_Check_Error(m01_rs1_r2.fan_diff_pres_error, bR2FanDiffPresError, CONCAT(_RS01, _R2), gsFanDiffPresSensorError, gsProcessWillContinue);
m01_rs1_r2.reactor_pres													:= F_AnalogIn(m01_rs1_r2.PT_01, m01_rs1_r2.reactor_pres_low, m01_rs1_r2.reactor_pres_high, m01_rs1_r2.reactor_pres_min, m01_rs1_r2.reactor_pres_offset);
bR2ReactorPresError														:= P_Alarms.M_Check_Error(m01_rs1_r2.reactor_pres_error, bR2ReactorPresError, CONCAT(_RS01, _R2), gsReactorPresSensorError, gsProcessWillContinue);
R_S.R2_reactor_pres														:= m01_rs1_r2.reactor_pres;
R_S.R2_reactor_pres_error												:= bR2ReactorPresError;
bR2OverMaxPressure														:= NOT m01_rs1_r2.reactor_pres_error AND m01_rs1_r2.reactor_pres > m01.SP_maximum_safe_reactor_steam_pressure;

m01_rs1_r3.inlet_co2													:= F_AnalogIn(m01_rs1_r3.AT_01, m01_rs1_r3.inlet_co2_low, m01_rs1_r3.inlet_co2_high, m01_rs1_r3.inlet_co2_min, m01_rs1_r3.inlet_co2_offset);
bR3InletCO2Error														:= P_Alarms.M_Check_Error(m01_rs1_r3.inlet_co2_error, bR3InletCO2Error, CONCAT(_RS01, _R3), gsInletCO2SensorError, gsProcessWillContinue);
m01_rs1_r3.inlet_h2o													:= F_AnalogIn(m01_rs1_r3.AT_02, m01_rs1_r3.inlet_h2o_low, m01_rs1_r3.inlet_h2o_high, m01_rs1_r3.inlet_h2o_min, m01_rs1_r3.inlet_h2o_offset);
bR3InletH2OError														:= P_Alarms.M_Check_Error(m01_rs1_r3.inlet_h2o_error, bR3InletH2OError, CONCAT(_RS01, _R3), gsInletH2OSensorError, gsProcessWillContinue);
m01_rs1_r3.outlet_co2													:= F_AnalogIn(m01_rs1_r3.AT_03, m01_rs1_r3.outlet_co2_low, m01_rs1_r3.outlet_co2_high, m01_rs1_r3.outlet_co2_min, m01_rs1_r3.outlet_co2_offset);
bR3OutletCO2Error														:= P_Alarms.M_Check_Error(m01_rs1_r3.outlet_co2_error, bR3OutletCO2Error, CONCAT(_RS01, _R3), gsOutletCO2SensorError, gsProcessWillContinue);
m01_rs1_r3.outlet_h2o													:= F_AnalogIn(m01_rs1_r3.AT_04, m01_rs1_r3.outlet_h2o_low, m01_rs1_r3.outlet_h2o_high, m01_rs1_r3.outlet_h2o_min, m01_rs1_r3.outlet_h2o_offset);
bR3OutletH2OError														:= P_Alarms.M_Check_Error(m01_rs1_r3.outlet_h2o_error, bR3OutletH2OError, CONCAT(_RS01, _R3), gsOutletH2OSensorError, gsProcessWillContinue);
m01_rs1_r3.air_flow														:= F_AnalogIn(m01_rs1_r3.FT_01, m01_rs1_r3.air_flow_low, m01_rs1_r3.air_flow_high, m01_rs1_r3.air_flow_min, m01_rs1_r3.air_flow_offset);
bR3AirFlowError															:= P_Alarms.M_Check_Error(m01_rs1_r3.air_flow_error, bR3AirFlowError, CONCAT(_RS01, _R3), gsAirFlowSensorError, gsProcessWillContinue);
m01_rs1_r3.filter_diff_pres												:= F_AnalogIn(m01_rs1_r3.PDT_01, m01_rs1_r3.filter_diff_pres_low, m01_rs1_r3.filter_diff_pres_high, m01_rs1_r3.filter_diff_pres_min, m01_rs1_r3.filter_diff_pres_offset);
bR3FilterDiffPresError													:= P_Alarms.M_Check_Error(m01_rs1_r3.filter_diff_pres_error, bR3FilterDiffPresError, CONCAT(_RS01, _R3), gsFilterDiffPresSensorError, gsProcessWillContinue);
m01_rs1_r3.sorbent_diff_pres											:= F_AnalogIn(m01_rs1_r3.PDT_02, m01_rs1_r3.sorbent_diff_pres_low, m01_rs1_r3.sorbent_diff_pres_high, m01_rs1_r3.sorbent_diff_pres_min, m01_rs1_r3.sorbent_diff_pres_offset,);
bR3SorbentDiffPresError													:= P_Alarms.M_Check_Error(m01_rs1_r3.sorbent_diff_pres_error, bR3SorbentDiffPresError, CONCAT(_RS01, _R3), gsSorbentDiffPresSensorError, gsProcessWillContinue);
m01_rs1_r3.fan_diff_pres												:= F_AnalogIn(m01_rs1_r3.PDT_03, m01_rs1_r3.fan_diff_pres_low, m01_rs1_r3.fan_diff_pres_high, m01_rs1_r3.fan_diff_pres_min, m01_rs1_r3.fan_diff_pres_offset);
bR3FanDiffPresError														:= P_Alarms.M_Check_Error(m01_rs1_r3.fan_diff_pres_error, bR3FanDiffPresError, CONCAT(_RS01, _R3), gsFanDiffPresSensorError, gsProcessWillContinue);
m01_rs1_r3.reactor_pres													:= F_AnalogIn(m01_rs1_r3.PT_01, m01_rs1_r3.reactor_pres_low, m01_rs1_r3.reactor_pres_high, m01_rs1_r3.reactor_pres_min, m01_rs1_r3.reactor_pres_offset);
bR3ReactorPresError														:= P_Alarms.M_Check_Error(m01_rs1_r3.reactor_pres_error, bR3ReactorPresError, CONCAT(_RS01, _R3), gsReactorPresSensorError, gsProcessWillContinue);
R_S.R3_reactor_pres														:= m01_rs1_r3.reactor_pres;
R_S.R3_reactor_pres_error												:= bR3ReactorPresError;
bR3OverMaxPressure														:= NOT m01_rs1_r3.reactor_pres_error AND m01_rs1_r3.reactor_pres > m01.SP_maximum_safe_reactor_steam_pressure;

m01_rs1_r4.inlet_co2													:= F_AnalogIn(m01_rs1_r4.AT_01, m01_rs1_r4.inlet_co2_low, m01_rs1_r4.inlet_co2_high, m01_rs1_r4.inlet_co2_min, m01_rs1_r4.inlet_co2_offset);
bR4InletCO2Error														:= P_Alarms.M_Check_Error(m01_rs1_r4.inlet_co2_error, bR4InletCO2Error, CONCAT(_RS01, _R4), gsInletCO2SensorError, gsProcessWillContinue);
m01_rs1_r4.inlet_h2o													:= F_AnalogIn(m01_rs1_r4.AT_02, m01_rs1_r4.inlet_h2o_low, m01_rs1_r4.inlet_h2o_high, m01_rs1_r4.inlet_h2o_min, m01_rs1_r4.inlet_h2o_offset);
bR4InletH2OError														:= P_Alarms.M_Check_Error(m01_rs1_r4.inlet_h2o_error, bR4InletH2OError, CONCAT(_RS01, _R4), gsInletH2OSensorError, gsProcessWillContinue);
m01_rs1_r4.outlet_co2													:= F_AnalogIn(m01_rs1_r4.AT_03, m01_rs1_r4.outlet_co2_low, m01_rs1_r4.outlet_co2_high, m01_rs1_r4.outlet_co2_min, m01_rs1_r4.outlet_co2_offset);
bR4OutletCO2Error														:= P_Alarms.M_Check_Error(m01_rs1_r4.outlet_co2_error, bR4OutletCO2Error, CONCAT(_RS01, _R4), gsOutletCO2SensorError, gsProcessWillContinue);
m01_rs1_r4.outlet_h2o													:= F_AnalogIn(m01_rs1_r4.AT_04, m01_rs1_r4.outlet_h2o_low, m01_rs1_r4.outlet_h2o_high, m01_rs1_r4.outlet_h2o_min, m01_rs1_r4.outlet_h2o_offset);
bR4OutletH2OError														:= P_Alarms.M_Check_Error(m01_rs1_r4.outlet_h2o_error, bR4OutletH2OError, CONCAT(_RS01, _R4), gsOutletH2OSensorError, gsProcessWillContinue);
m01_rs1_r4.air_flow														:= F_AnalogIn(m01_rs1_r4.FT_01, m01_rs1_r4.air_flow_low, m01_rs1_r4.air_flow_high, m01_rs1_r4.air_flow_min, m01_rs1_r4.air_flow_offset);
bR4AirFlowError															:= P_Alarms.M_Check_Error(m01_rs1_r4.air_flow_error, bR4AirFlowError, CONCAT(_RS01, _R4), gsAirFlowSensorError, gsProcessWillContinue);
m01_rs1_r4.filter_diff_pres												:= F_AnalogIn(m01_rs1_r4.PDT_01, m01_rs1_r4.filter_diff_pres_low, m01_rs1_r4.filter_diff_pres_high, m01_rs1_r4.filter_diff_pres_min, m01_rs1_r4.filter_diff_pres_offset);
bR4FilterDiffPresError													:= P_Alarms.M_Check_Error(m01_rs1_r4.filter_diff_pres_error, bR4FilterDiffPresError, CONCAT(_RS01, _R4), gsFilterDiffPresSensorError, gsProcessWillContinue);
m01_rs1_r4.sorbent_diff_pres											:= F_AnalogIn(m01_rs1_r4.PDT_02, m01_rs1_r4.sorbent_diff_pres_low, m01_rs1_r4.sorbent_diff_pres_high, m01_rs1_r4.sorbent_diff_pres_min, m01_rs1_r4.sorbent_diff_pres_offset,);
bR4SorbentDiffPresError													:= P_Alarms.M_Check_Error(m01_rs1_r4.sorbent_diff_pres_error, bR4SorbentDiffPresError, CONCAT(_RS01, _R4), gsSorbentDiffPresSensorError, gsProcessWillContinue);
m01_rs1_r4.fan_diff_pres												:= F_AnalogIn(m01_rs1_r4.PDT_03, m01_rs1_r4.fan_diff_pres_low, m01_rs1_r4.fan_diff_pres_high, m01_rs1_r4.fan_diff_pres_min, m01_rs1_r4.fan_diff_pres_offset);
bR4FanDiffPresError														:= P_Alarms.M_Check_Error(m01_rs1_r4.fan_diff_pres_error, bR4FanDiffPresError, CONCAT(_RS01, _R4), gsFanDiffPresSensorError, gsProcessWillContinue);
m01_rs1_r4.reactor_pres													:= F_AnalogIn(m01_rs1_r4.PT_01, m01_rs1_r4.reactor_pres_low, m01_rs1_r4.reactor_pres_high, m01_rs1_r4.reactor_pres_min, m01_rs1_r4.reactor_pres_offset);
bR4ReactorPresError														:= P_Alarms.M_Check_Error(m01_rs1_r4.reactor_pres_error, bR4ReactorPresError, CONCAT(_RS01, _R4), gsReactorPresSensorError, gsProcessWillContinue);
R_S.R4_reactor_pres														:= m01_rs1_r4.reactor_pres;
R_S.R4_reactor_pres_error												:= bR4ReactorPresError;
bR4OverMaxPressure														:= NOT m01_rs1_r4.reactor_pres_error AND m01_rs1_r4.reactor_pres > m01.SP_maximum_safe_reactor_steam_pressure;

rAveragePressure														:= 0;
iCount																	:= 0;
iVacuumStatus															:= 0;
iError																	:= 4;
IF NOT m01_rs1_r1.reactor_pres_error THEN
	rAveragePressure													:= rAveragePressure + m01_rs1_r1.reactor_pres;
	iVacuumStatus														:= F_LowMidHigh(m01_rs1_r1.reactor_pres, m01.SP_target_desorption_starting_pressure, m01.SP_maximum_desorption_starting_pressure, iVacuumStatus);
	iCount																:= iCount + 1;
	iError																:= iError - 1;
END_IF
IF NOT m01_rs1_r2.reactor_pres_error THEN
	rAveragePressure													:= rAveragePressure + m01_rs1_r2.reactor_pres;
	iVacuumStatus														:= F_LowMidHigh(m01_rs1_r2.reactor_pres, m01.SP_target_desorption_starting_pressure, m01.SP_maximum_desorption_starting_pressure, iVacuumStatus);
	iCount																:= iCount + 1;
	iError																:= iError - 1;
END_IF
IF NOT m01_rs1_r3.reactor_pres_error THEN
	rAveragePressure													:= rAveragePressure + m01_rs1_r3.reactor_pres;
	iVacuumStatus														:= F_LowMidHigh(m01_rs1_r3.reactor_pres, m01.SP_target_desorption_starting_pressure, m01.SP_maximum_desorption_starting_pressure, iVacuumStatus);
	iCount																:= iCount + 1;
	iError																:= iError - 1;
END_IF
IF NOT m01_rs1_r4.reactor_pres_error THEN
	rAveragePressure													:= rAveragePressure + m01_rs1_r4.reactor_pres;
	iVacuumStatus														:= F_LowMidHigh(m01_rs1_r1.reactor_pres, m01.SP_target_desorption_starting_pressure, m01.SP_maximum_desorption_starting_pressure, iVacuumStatus);
	iCount																:= iCount + 1;
	iError																:= iError - 1;
END_IF

R_S.average_reactor_pressure											:= SEL(iCount > 0, 0, rAveragePressure / iCount);
R_S.reactor_pressure_error												:= SEL(iError >= _MAX_REACTOR_ERRORS, '', F_Concat3(INT_TO_STRING(iError), ' ', gsReactorPresError));
R_S.reactor_vacuum_status												:= iVacuumStatus;
average_pressure_within_ambient											:= rAveragePressure >= P_M01.rMinPressureSP AND rAveragePressure <= P_M01.rMaxPressureSP;
R_S.average_reactor_pressure_within_ambient								:= average_pressure_within_ambient;
fb_RS_IO.reactor_over_max_pressure										:= bR1OverMaxPressure OR bR2OverMaxPressure OR bR3OverMaxPressure OR bR4OverMaxPressure;

R_S.R1_inlet_co2														:= m01_rs1_r1.inlet_co2;

R_S.R1_outlet_co2														:= m01_rs1_r1.outlet_co2;

ACTION A_Reactor_Set:
// Phase 0 - P_M01_RS01.A_Reactor_Set
// Rev 1.0 - May 10, 2024

fb_RS(		U															:= P_U01.u,
			R_S															:= P_M01_RS01.R_S,
			Stop_Reactor_Set											:= stop_reactor_set,
			Clear_Reactor_Set_Pause										:= clear_reactor_set_pause,
			test_error													:= gbRS01TestError,									///@@@ Temporary for testing
			RS_Name														:= _RS01,
			RS_Number													:= 1,
			Cycle_Mode													:= P_M01.sCycleModeRS01,
			Fan_Setpoint												:= m01.SP_reactor_set_1_vfd_percent,
//			Evac_Service_Acked											:= P_M01.evac_service_acked,
			Evac_Service_Assigned										:= P_M01.evac_service_assigned[1],
			Steam_Service_Assigned										:= P_M01.steam_service_assigned[1],
			Cycle_Stage													=> gsM01RS01CycleStage,
			Remaining_Time												=> m01_rs1.tr_Remaining_Time,
			Current_Step												=> m01_rs1.ti_Current_Step,
			Machine_State												=> m01_rs1.ti_Machine_State,
			Status														=> m01_rs1.ti_Status,
			Process_Running												=> m01_rs1.tb_Process_Running,
			Repressurization_Running									=> m01_rs1.tb_Repressurization_Running,
			Adsorption_Running											=> m01_rs1.tb_Adsorption_Running,
			Evacuation_Running											=> m01_rs1.tb_Evacuation_Running,
			Desorption_Running											=> m01_rs1.tb_Desorption_Running,
			Process_Complete											=> m01_rs1.tb_Process_Complete,
			Utility_Error												=> utility_error,
			Stop_M01_RS													=> stop_rs_automode,
			Cancel_Reactor_Set											=> cancel_reactor_set,
			Cancel_All_Reactor_Sets										=> cancel_all_reactor_sets,
			Done														=> reactor_done);

fb_RS_IO(	power_control_in											:= m01_rs1.power_control,
			power_control_out											=> m01_rs1.power_control_status,
			PWR_01														=> m01_rs1.PWR_01,
			power_control_fdbk_no										:= m01_rs1.circuit_breaker_no_feedback,
			power_control_fdbk_nc										:= m01_rs1.circuit_breaker_nc_feedback,
			condensate_lsl_in											:= m01_rs1.condensate_lsl,
			condensate_lsh_in											:= m01_rs1.condensate_lsh,
			condensate_lsl_out											=> R_S.condensate_lsl,
			condensate_lsh_out											=> R_S.condensate_lsh,
			condensate_pump_hmi											:= m01_rs1.condensate_pump,
			condensate_pump_plc											:= R_S.condensate_pump,
			condensate_pump_cmd_status									=> m01_rs1.condensate_pump_cmd_status,
			P_01														=> m01_rs1.P_01,
			rs_close_valves												:= R_S.close_all_valves,
			dead_air_valve_hmi											:= m01_rs1.dead_air_valve,
			dead_air_valve_plc											:= R_S.dead_air_valve,
			dead_air_valve_open_cmd_status								=> m01_rs1.dead_air_valve_open_cmd_status,
			dead_air_valve_open											:= m01_rs1.dead_air_valve_open,
			dead_air_valve_closed										:= m01_rs1.dead_air_valve_closed,
			dead_air_valve_clear										=> R_S.dead_air_valve_clear,
			XV_04														=> m01_rs1.XV_04,
			purge_valve_hmi												:= m01_rs1.purge_valve,
			purge_valve_plc												:= R_S.purge_valve,
			purge_valve_open_cmd_status									=> m01_rs1.purge_valve_open_cmd_status,
			purge_valve_open											:= m01_rs1.purge_valve_open,
			purge_valve_closed											:= m01_rs1.purge_valve_closed,
			purge_valve_clear											=> R_S.purge_valve_clear, 
			XV_05														=> m01_rs1.XV_05,
			cooling_valve_hmi											:= m01_rs1.cooling_valve,
			cooling_valve_plc											:= R_S.cooling_valve,
			cooling_valve_open_cmd_status								=> m01_rs1.cooling_valve_open_cmd_status,
			cooling_valve_open											:= m01_rs1.cooling_valve_open,
			cooling_valve_closed										:= m01_rs1.cooling_valve_closed,
			cooling_valve_clear											=> R_S.cooling_valve_clear,
			XV_06														=> m01_rs1.XV_06,
			steam_header_valve_hmi										:= m01_rs1.steam_header_valve,
			steam_header_valve_plc										:= R_S.steam_header_valve,
			steam_header_valve_open_cmd_status							=> m01_rs1.steam_header_valve_open_cmd_status,
			steam_header_valve_open										:= m01_rs1.steam_header_valve_open,
			steam_header_valve_closed									:= m01_rs1.steam_header_valve_closed,
			steam_header_valve_not_closed								=> R_S.steam_header_valve_not_closed,
			steam_header_valve_clear									=> R_S.steam_header_valve_clear,
			XV_07														=> m01_rs1.XV_07,
			steam_control_valve_hmi										:= m01_rs1.steam_control_valve,
			steam_control_valve_plc										:= R_S.steam_control_valve,
			steam_control_valve_mode_hmi								:= m01_rs1.steam_control_valve_mode,
			steam_control_valve_mode_plc								:= R_S.steam_control_valve_mode,
			steam_control_valve_current_mode							=> m01_rs1.steam_control_valve_current_mode,
			steam_control_valve_error									:= m01_rs1.steam_control_valve_position_error,
			steam_control_valve_position								=> R_S.steam_control_valve_position,
			steam_control_valve_closed									=> R_S.steam_control_valve_closed,			
			steam_control_valve_setpoint								:= R_S.steam_control_valve_setpoint,
			steam_control_valve_control_point							:= R_S.steam_control_valve_control_point,
			steam_control_valve_loop_time								:= m01_rs1.steam_control_valve_loop_time,
			steam_control_valve_kp										:= m01_rs1.steam_control_valve_kp,
			steam_control_valve_ki										:= m01_rs1.steam_control_valve_ki,
			steam_control_valve_iband									:= m01_rs1.steam_control_valve_iband,
			steam_control_valve_base									:= m01_rs1.steam_control_valve_base,
			steam_control_valve_base_adjust								:= m01_rs1.steam_control_valve_base_adjust,
			PCV_01														=> m01_rs1.PCV_01,
			status_in													:= m01_rs1.ti_Status,
			status_out													=> m01_rs1.ts_Status_Text,
			valves_clear												=> R_S.valves_clear);
END_ACTION

ACTION A_Reactor1_IO:
// Phase 0 - P_M01_RS01.A_Reactor1_IO
// Rev 1.0 - April 26, 2024

fb_R1_IO(	RSet														:= _RS01,
			React														:= _R1,
			
			Power_On													:= m01_rs1.power_control,
			                                                    
			sorbent_low_temp											=> m01_rs1_r1.temp_low,
			sorbent_high_temp											=> m01_rs1_r1.temp_high,
			sorbent_average_temp										=> m01_rs1_r1.temp_average,
			                                                    
